	  //  // Brak przepływu na powrocie
	    
	  //   #nr := 7;
	  //   CASE "Tor1_alarmy".alarm[#nr].procedura OF
	            
	  //       2: //zalacz
	  //           IF "Tor1_obiekty".obiekt["C101FV11"].hmiPotwWysterowania =0 AND ("Tor1_hmi".button.bPauza.set=0)
	                
	                
	  //           THEN
	  //               IF "Tor1_alarmy".alarm[#nr].timerek < 32000 THEN
	  //                   "Tor1_alarmy".alarm[#nr].timerek := "Tor1_alarmy".alarm[#nr].timerek + 1;
	  //               END_IF;
	  //               "Tor1_alarmy".alarm[#nr].stan := BOOL_TO_INT("Tor1_alarmy".alarm[#nr].timerek >
	  //               "Tor1_RecepturyStacjaMycia".Receptura[#aktualnyNumerReceptury].Krok[#aktualnyKrokMycia].PM[4] * 10);
	  //           ELSE
	  //               "Tor1_alarmy".alarm[#nr].timerek := 0;
	  //               "Tor1_alarmy".alarm[#nr].stan := 0;
	  //           END_IF;
	            
	  //           IF "Tor1_alarmy".alarm[#nr].stan = 1
	  //               AND "Tor1_program".program.numerKroku <> 7700 THEN
	  //               "Tor1_hmi".button.bPauza.set := 1;
	  //               "krokZapauzowany" := "Tor1_program".program.numerKroku;
	  //               "Tor1_program".program.numerKroku := 7700;
	  //           END_IF;
	            
	  //       0:
	  //           "Tor1_alarmy".alarm[#nr].timerek := 0;
	  //           "Tor1_alarmy".alarm[#nr].stan := 0;
	            
	  //   END_CASE;
	    
	    
	    
	  //   //Niskie stężenie ługu
	    
	  //   #nr :=8;
	  //   CASE "Tor1_alarmy".alarm[#nr].procedura OF
	            
	  //       2: //zalacz
	  //           IF "Tor1_obiekty".obiekt["C101CT11"].WartośćPomiaru <=
	  //               0.5 * "Tor1_RecepturyStacjaMycia".Receptura[#aktualnyNumerReceptury].Krok[#aktualnyKrokMycia].PM[10]
	  //               AND #aktualnyKrokMycia=3
	                
	  //           THEN
	  //               IF "Tor1_alarmy".alarm[#nr].timerek < 32000 THEN
	  //                   "Tor1_alarmy".alarm[#nr].timerek := "Tor1_alarmy".alarm[#nr].timerek + 1;
	  //               END_IF;
	  //               "Tor1_alarmy".alarm[#nr].stan := BOOL_TO_INT("Tor1_alarmy".alarm[#nr].timerek >600);
	  //           ELSE
	  //               "Tor1_alarmy".alarm[#nr].timerek := 0;
	  //               "Tor1_alarmy".alarm[#nr].stan := 0;
	  //           END_IF;
	        
	            
	  //   END_CASE;
	    
	    
	    
	    
	  //   //Niskie stężenie kwasu
	    
	  //   #nr := 9;
	  //   CASE "Tor1_alarmy".alarm[#nr].procedura OF
	            
	  //       2: //zalacz
	  //           IF "Tor1_obiekty".obiekt["C101CT11"].WartośćPomiaru <=
	  //               0.5 * "Tor1_RecepturyStacjaMycia".Receptura[#aktualnyNumerReceptury].Krok[#aktualnyKrokMycia].PM[10]
	  //               AND #aktualnyKrokMycia=4
	                
	  //           THEN
	  //               IF "Tor1_alarmy".alarm[#nr].timerek < 32000 THEN
	  //                   "Tor1_alarmy".alarm[#nr].timerek := "Tor1_alarmy".alarm[#nr].timerek + 1;
	  //               END_IF;
	  //               "Tor1_alarmy".alarm[#nr].stan := BOOL_TO_INT("Tor1_alarmy".alarm[#nr].timerek > 600);
	  //           ELSE
	  //               "Tor1_alarmy".alarm[#nr].timerek := 0;
	  //               "Tor1_alarmy".alarm[#nr].stan := 0;
	  //           END_IF;
	            
	       
	            
	  //   END_CASE;
	    
	    
	  //   //Brak stężonego ługu
	    
	  //   #nr := 10;
	  //   CASE "Tor1_alarmy".alarm[#nr].procedura OF
	            
	  //       2: //zalacz
	  //           IF "CIP0_obiekty".obiekt["C2L1LL01"].hmiPotwWysterowania = 0
	                
	                
	                
	  //           THEN
	  //               IF "Tor1_alarmy".alarm[#nr].timerek < 32000 THEN
	  //                   "Tor1_alarmy".alarm[#nr].timerek := "Tor1_alarmy".alarm[#nr].timerek + 1;
	  //               END_IF;
	  //               "Tor1_alarmy".alarm[#nr].stan := BOOL_TO_INT("Tor1_alarmy".alarm[#nr].timerek > 600);
	  //           ELSE
	  //               "Tor1_alarmy".alarm[#nr].timerek := 0;
	  //               "Tor1_alarmy".alarm[#nr].stan := 0;
	  //           END_IF;
	            
	          
	            
	  //   END_CASE;
	    
	  //   //Brak stężonego kwasu
	    
	  //   #nr := 11;
	  //   CASE "Tor1_alarmy".alarm[#nr].procedura OF
	            
	  //       2: //zalacz
	  //           IF "CIP0_obiekty".obiekt["C2A1LL01"].hmiPotwWysterowania = 0
	                
	                
	                
	  //           THEN
	  //               IF "Tor1_alarmy".alarm[#nr].timerek < 32000 THEN
	  //                   "Tor1_alarmy".alarm[#nr].timerek := "Tor1_alarmy".alarm[#nr].timerek + 1;
	  //               END_IF;
	  //               "Tor1_alarmy".alarm[#nr].stan := BOOL_TO_INT("Tor1_alarmy".alarm[#nr].timerek > 600);
	  //           ELSE
	  //               "Tor1_alarmy".alarm[#nr].timerek := 0;
	  //               "Tor1_alarmy".alarm[#nr].stan := 0;
	  //           END_IF;
	    
	            
	  //   END_CASE;
	    
	    //Brak dezynfekanta
	    
	    #nr := 12;
	    CASE "Tor1_alarmy".alarm[#nr].procedura OF
	            
	        2: //zalacz
	            IF                "Cip".obiekt["Cip".tor[1].zbiorniczekDozowanieDezynfekantu.czujnikDolnegoPoziomu].hmiPotwWysterowania=0
	                OR (  "Cip".obiekt["Cip".tor[1].czujnikPrzepływuDozowanegoDezynfekantu].hmiPotwWysterowania=0
	                AND "Cip".obiekt["Cip".tor[1].zawórDozowaniaDezynfekantuwLinię].hmiPotwWysterowania=1)
	                
	            THEN
	                IF "Tor1_alarmy".alarm[#nr].timerek < 32000 THEN
	                    "Tor1_alarmy".alarm[#nr].timerek := "Tor1_alarmy".alarm[#nr].timerek + 1;
	                END_IF;
	                "Tor1_alarmy".alarm[#nr].stan := BOOL_TO_INT("Tor1_alarmy".alarm[#nr].timerek > 600);
	            ELSE
	                "Tor1_alarmy".alarm[#nr].timerek := 0;
	                "Tor1_alarmy".alarm[#nr].stan := 0;
	            END_IF;
	         
	    END_CASE;
	    
	    
	        
	  //       #nr := 13;
	  //       CASE "Tor1_alarmy".alarm[#nr].procedura OF
	                
	  //           2: //zalacz
	  //               IF  "Tor1_program".program.opóżnienie
	  //                   >"Tor1_RecepturyStacjaMycia".Receptura[#aktualnyNumerReceptury].Krok[#aktualnyKrokMycia].PM[19]
	                    
	                    
	  //               THEN
	  //                   IF "Tor1_alarmy".alarm[#nr].timerek < 32000 THEN
	  //                       "Tor1_alarmy".alarm[#nr].timerek := "Tor1_alarmy".alarm[#nr].timerek + 1;
	  //                   END_IF;
	  //                   "Tor1_alarmy".alarm[#nr].stan := BOOL_TO_INT("Tor1_alarmy".alarm[#nr].timerek > 600);
	  //               ELSE
	  //                   "Tor1_alarmy".alarm[#nr].timerek := 0;
	  //                   "Tor1_alarmy".alarm[#nr].stan := 0;
	  //               END_IF;
	         
	                
	  //       END_CASE;
	  
END_FUNCTION

FUNCTION "Tor1.procedury_obiektów" : Void
{ S7_Optimized_Access := 'TRUE' }
VERSION : 0.1
   VAR_TEMP 
      obj : Int;
      nr : Int;
      Mnr : String;
      aktualnyNumerReceptury : Int;
      aktualnyKrokMycia : Int;
      temp : Int;
   END_VAR


BEGIN
	    //program zawiera procedury dla napedów i zaworów dla procedur o numerze >1  (procedura 0 i 1 jest obsługiwana w programie Obsługa obiektów)
	    //procedury wyzwalane  z progrmu TablicaProcedór dla kolejnych kroków  "F1".obiekt["F100CP01"].procedura: = 2
	    //wyzwolenie procedury zero  automatycznie  wyłącza naped/zawór
	    //procedura:=1   uruchamia napęd/zawór na 100% - czyli załaczenie napedu jak kiedyś SET -- obsługiwana jest w programie Obsługa obiektów
	    //PAUZA może być obsługiwana w każdej procedurze z osobna
	    //
	    //open ctrl+shift+(*)Numeric
	    //close ctrl+shift+(/)Numeric
	    
	    #aktualnyNumerReceptury := "Tor1_RecepturyStacjaMycia".numerUżywanejReceptury;
	    #aktualnyKrokMycia := "Tor1_RecepturyStacjaMycia".numerKrokuMycia;
	    #temp := "Tor1_program".program.numerKroku;
	    
	    REGION POMPA PODAWANIA CIP
	    
	    #nr := "Cip".tor[1].pompaPodawaniaCip;
	    CASE "Tor1_program".program.numerKroku OF
	    7210, 7220, 7250:
	    "Cip".obiekt[#nr].procedura := 2;
	    7244, 7270, 7281..7287,7310, 7320,7321, 7414, 7420:
	    "Cip".obiekt[#nr].procedura := 3;
	    7240, 7242, 7243, 7246:
	    "Cip".obiekt[#nr].procedura := 6;
	    7100:
	    "Cip".obiekt[#nr].procedura := 7;
	    ELSE
	    "Cip".obiekt[#nr].procedura := 0;
	    
	    END_CASE;
	    
	    
	    
	    CASE "Cip".obiekt[#nr].procedura OF
	    2:
	    //wyzwolenie timerków
	    "Cip".obiekt[#nr].SetReset.czasDoSet := 3;
	    "Cip".obiekt[#nr].SetReset.inSet := "Cip".obiekt["Cip".tor[0].zbiornikwodyCzystej.czujnikDolnegoPoziomu].hmiPotwWysterowania
	    OR "Cip".obiekt["Cip".tor[0].zbiornikWodyWtórnej.czujnikDolnegoPoziomu].hmiPotwWysterowania;
	    "Cip".obiekt[#nr].SetReset.czasDoReset := 5;
	    "Cip".obiekt[#nr].SetReset.inReset := (NOT "Cip".obiekt["Cip".tor[0].zbiornikwodyCzystej.czujnikDolnegoPoziomu].hmiPotwWysterowania
	    AND NOT "Cip".obiekt["Cip".tor[0].zbiornikWodyWtórnej.czujnikDolnegoPoziomu].hmiPotwWysterowania) OR
	    ("Cip".obiekt["Cip".tor[1].zbiornikDezynfekantu.czujnikDolnegoPoziomu].hmiPotwWysterowania = 0 AND ("Tor1_program".program.numerKroku = 7282
	    OR "Tor1_program".program.numerKroku = 7283))
	    
	    ;
	    
	    //załaczanie
	    "Cip".obiekt[#nr].inStartAuto := "Cip".obiekt[#nr].SetReset.wyjście;
	    
	    //wysterowanie
	    "Cip".obiekt[#nr].inZadaneWysterowanieAuto :=  //pid_out wypełniamy w wywołaniu pida z out pida
	    LIMIT(IN := "Cip".obiekt[#nr].pid_Out, MN := 0.0, MX := 100.0);//pid_out ;
	    
	    ////PID
	    "Cip".obiekt[#nr].pid_SP := "Tor1_RecepturyStacjaMycia".Receptura[#aktualnyNumerReceptury].Krok[#aktualnyKrokMycia].PM[2];
	    "Cip".obiekt[#nr].pid_PV := "Cip".obiekt["Cip".tor[1].przepływomierzZaWymiennikiem].WartośćPomiaru;
	    
	    
	    3: //wyzwolenie timerków
	    
	    //wyzwolenie timerków
	    "Cip".obiekt[#nr].SetReset.czasDoSet := 3;
	    "Cip".obiekt[#nr].SetReset.inSet := "Cip".obiekt["Cip".tor[0].zbiornikwodyCzystej.czujnikDolnegoPoziomu].hmiPotwWysterowania
	    ;
	    "Cip".obiekt[#nr].SetReset.czasDoReset := 5;
	    "Cip".obiekt[#nr].SetReset.inReset := NOT "Cip".obiekt["Cip".tor[0].zbiornikwodyCzystej.czujnikDolnegoPoziomu].hmiPotwWysterowania
	    ;
	    //załaczanie
	    
	    "Cip".obiekt[#nr].inStartAuto := "Cip".obiekt[#nr].SetReset.wyjście;
	    
	    //wysterowanie
	    "Cip".obiekt[#nr].inZadaneWysterowanieAuto :=  //pid_out wypełniamy w wywołaniu pida z out pida
	    LIMIT(IN := "Cip".obiekt[#nr].pid_Out, MN := 0.0, MX := 100.0);//pid_out ;
	    
	    ////PID
	    "Cip".obiekt[#nr].pid_SP := "Tor1_RecepturyStacjaMycia".Receptura[#aktualnyNumerReceptury].Krok[#aktualnyKrokMycia].PM[2];
	    "Cip".obiekt[#nr].pid_PV := "Cip".obiekt["Cip".tor[1].przepływomierzZaWymiennikiem].WartośćPomiaru;
	    
	    4: //wyzwolenie timerków
	    
	    //wyzwolenie timerków
	    "Cip".obiekt[#nr].SetReset.czasDoSet := 3;
	    "Cip".obiekt[#nr].SetReset.inSet :=
	    "Cip".obiekt["Cip".tor[0].zbiornikwodyCzystej.czujnikDolnegoPoziomu].hmiPotwWysterowania
	    AND #aktualnyKrokMycia = 3
	    ;
	    "Cip".obiekt[#nr].SetReset.czasDoReset := 5;
	    "Cip".obiekt[#nr].SetReset.inReset :=
	    NOT "Cip".obiekt["Cip".tor[0].zbiornikwodyCzystej.czujnikDolnegoPoziomu].hmiPotwWysterowania
	    AND #aktualnyKrokMycia = 3
	    ;
	    //załaczanie
	    "Cip".obiekt[#nr].inStartAuto := "Cip".obiekt[#nr].SetReset.wyjście;
	    
	    //wysterowanie
	    "Cip".obiekt[#nr].inZadaneWysterowanieAuto :=  //pid_out wypełniamy w wywołaniu pida z out pida
	    LIMIT(IN := "Cip".obiekt[#nr].pid_Out, MN := 0.0, MX := 100.0);//pid_out ;
	    
	    ////PID
	    "Cip".obiekt[#nr].pid_SP := "Tor1_RecepturyStacjaMycia".Receptura[#aktualnyNumerReceptury].Krok[#aktualnyKrokMycia].PM[2];
	    "Cip".obiekt[#nr].pid_PV := "Cip".obiekt["Cip".tor[1].przepływomierzZaWymiennikiem].WartośćPomiaru;
	    
	    5: //wyzwolenie timerków
	    
	    //wyzwolenie timerków
	    "Cip".obiekt[#nr].SetReset.czasDoSet := 3;
	    "Cip".obiekt[#nr].SetReset.inSet := "Cip".obiekt["Cip".tor[0].zbiornikwodyCzystej.czujnikDolnegoPoziomu].hmiPotwWysterowania
	    AND #aktualnyKrokMycia = 4
	    ;
	    "Cip".obiekt[#nr].SetReset.czasDoReset := 5;
	    "Cip".obiekt[#nr].SetReset.inReset := NOT "Cip".obiekt["Cip".tor[0].zbiornikwodyCzystej.czujnikDolnegoPoziomu].hmiPotwWysterowania
	    AND #aktualnyKrokMycia = 4
	    ;
	    //załaczanie
	    "Cip".obiekt[#nr].inStartAuto := "Cip".obiekt[#nr].SetReset.wyjście;
	    
	    //wysterowanie
	    "Cip".obiekt[#nr].inZadaneWysterowanieAuto :=  //pid_out wypełniamy w wywołaniu pida z out pida
	    LIMIT(IN := "Cip".obiekt[#nr].pid_Out, MN := 0.0, MX := 100.0);//pid_out ;
	    
	    ////PID
	    "Cip".obiekt[#nr].pid_SP := "Tor1_RecepturyStacjaMycia".Receptura[#aktualnyNumerReceptury].Krok[#aktualnyKrokMycia].PM[2];
	    "Cip".obiekt[#nr].pid_PV := "Cip".obiekt["Cip".tor[1].przepływomierzZaWymiennikiem].WartośćPomiaru;
	    
	    6: //wyzwolenie timerków
	    //wyzwolenie timerków
	    "Cip".obiekt[#nr].SetReset.czasDoSet := 3;
	    "Cip".obiekt[#nr].SetReset.inSet :=
	    ("Cip".obiekt["Cip".tor[0].zbiornikwodyCzystej.czujnikDolnegoPoziomu].hmiPotwWysterowania
	    AND #aktualnyKrokMycia = 4)
	    OR
	    ("Cip".obiekt["Cip".tor[0].zbiornikwodyCzystej.czujnikDolnegoPoziomu].hmiPotwWysterowania
	    AND #aktualnyKrokMycia = 3)
	    ;
	    "Cip".obiekt[#nr].SetReset.czasDoReset := 5;
	    "Cip".obiekt[#nr].SetReset.inReset :=
	    (NOT "Cip".obiekt["Cip".tor[0].zbiornikwodyCzystej.czujnikDolnegoPoziomu].hmiPotwWysterowania
	    AND #aktualnyKrokMycia = 4)
	    OR
	    (NOT "Cip".obiekt["Cip".tor[0].zbiornikwodyCzystej.czujnikDolnegoPoziomu].hmiPotwWysterowania
	    AND #aktualnyKrokMycia = 3);
	    
	    //załaczanie
	    "Cip".obiekt[#nr].inStartAuto := 1;
	    
	    //wysterowanie
	    "Cip".obiekt[#nr].inZadaneWysterowanieAuto :=  //pid_out wypełniamy w wywołaniu pida z out pida
	    LIMIT(IN := "Cip".obiekt[#nr].pid_Out, MN := 0.0, MX := 100.0);//pid_out ;
	    
	    ////PID
	    "Cip".obiekt[#nr].pid_SP := "Tor1_RecepturyStacjaMycia".Receptura[#aktualnyNumerReceptury].Krok[#aktualnyKrokMycia].PM[2];
	    "Cip".obiekt[#nr].pid_PV := "Cip".obiekt["Cip".tor[1].przepływomierzZaWymiennikiem].WartośćPomiaru;
	    
	    
	    7:
	    //wyzwolenie timerków
	    "Cip".obiekt[#nr].SetReset.czasDoSet := 1;
	    "Cip".obiekt[#nr].SetReset.inSet :=
	    "Cip".obiekt["Cip".tor[2].pompaPodawaniaCip].inStartAuto; //cpNiex
	    
	    "Cip".obiekt[#nr].SetReset.czasDoReset := 1;
	    "Cip".obiekt[#nr].SetReset.inReset :=
	    NOT "Cip".obiekt["Cip".tor[2].pompaPodawaniaCip].inStartAuto; //cpNiex
	    //załaczanie
	    "Cip".obiekt[#nr].inStartAuto := "Cip".obiekt[#nr].SetReset.wyjście;
	    //wysterowanie
	    "Cip".obiekt[#nr].inZadaneWysterowanieAuto := 100.0;
	    
	    
	    
	    0:
	    ;
	    
	    // resetowanie całkującej części regulatora aby nie przejebać temperatury
	    // "PID_Compact23".IntegralResetMode := 3;
	    // "PID_Compact23".OverwriteInitialOutputValue := "F1.SP"."203"- 1.0;
	    // "PID_Compact23".Reset := "F1".obiekt["F100LT01"].WartośćPomiaru > 70.0;
	    // := LIMIT(IN := "APA".obiekt["PID123"].outWysterowanieUrządzenia,
	    // MN := 0.0, MX := "APA".obiekt["H101TT01"].WartośćPomiaru + "H1.STP"."214");
	    
	    END_CASE;
	    
	    IF "Cip".obiekt[#nr].procedura > 0 THEN
	    
	        IF "Cip".obiekt[#nr].inStartAuto = 0 THEN
	            "Cip".obiekt[#nr].inZadaneWysterowanieAuto := 0.0;
	            "Cip".obiekt[#nr].pid_SP := 0.0;
	        END_IF;
	    END_IF;
	    
	    
	    "PID.pompaPodawaniaCipTor1"(Setpoint := "Cip".obiekt[#nr].pid_SP,
	                        Input := "Cip".obiekt[#nr].pid_PV,
	                        Reset := "Cip".obiekt[#nr].hmiResetAwaria,
	                        Output => "Cip".obiekt[#nr].pid_Out);
	    "PID.pompaPodawaniaCipTor1".Retain.CtrlParams.Gain := 1.2;
	    "PID.pompaPodawaniaCipTor1".Retain.CtrlParams.Ti := 3;
	    "PID.pompaPodawaniaCipTor1".Retain.CtrlParams.Td := 0.1;
	    
	    
	    
	    "PID.pompaPodawaniaCipTor1".IntegralResetMode := 3;
	    "PID.pompaPodawaniaCipTor1".OverwriteInitialOutputValue := 1;
	    "PID.pompaPodawaniaCipTor1".Reset := (
	    "Cip".obiekt[#nr].procedura = 0 OR "Cip".obiekt[#nr].inStartAuto = 0
	    OR "numer_kroku_stary_1" <> "Tor1_program".program.numerKroku);
	    
	    "numer_kroku_stary_1" := "Tor1_program".program.numerKroku;
	    END_REGION
	    
	    REGION POMPA PRZYGOTOWANIA CIP(DRUGA PODAWCZA)
	    
	    //pompa powrotu/ Program musi ustalić, który tor myje stacje,
	    //drugi staje się pompą powrotu (staje się pompą 102 - tymczasowo)
	    //obsługa wykrywania w CIP1_wejściach_wyjściach
	    #nr := "Cip".tor[2].pompaPodawaniaCip;
	    CASE "Tor1_program".program.numerKroku OF
	    7401..7404, 7410..7414:
	    "Cip".obiekt[#nr].procedura := 2
	    ;
	    7230..7440:
	    "Cip".obiekt[#nr].procedura := 3;
	    7450, 7460:
	    "Cip".obiekt[#nr].procedura := 4;
	    ELSE
	    "Cip".obiekt[#nr].procedura := 0;
	    
	    END_CASE;
	    
	    
	    CASE "Cip".obiekt[#nr].procedura OF
	    2:
	    //wyzwolenie timerków
	    "Cip".obiekt[#nr].SetReset.czasDoSet := 3;
	    "Cip".obiekt[#nr].SetReset.inSet :=
	    "Cip".obiekt["Cip".tor[0].zbiornikWodyWtórnej.czujnikDolnegoPoziomu].hmiPotwWysterowania;
	    
	    "Cip".obiekt[#nr].SetReset.czasDoReset := 60;
	    "Cip".obiekt[#nr].SetReset.inReset :=
	    NOT "Cip".obiekt["Cip".tor[0].zbiornikWodyWtórnej.czujnikDolnegoPoziomu].hmiPotwWysterowania;
	    //załaczanie
	    
	    "Cip".obiekt[#nr].inStartAuto := "Cip".obiekt[#nr].SetReset.wyjście;
	    
	    //wysterowanie
	    "Cip".obiekt[#nr].inZadaneWysterowanieAuto := 100.0;
	    
	    3:
	    //wyzwolenie timerków
	    "Cip".obiekt[#nr].SetReset.czasDoSet := 3;
	    "Cip".obiekt[#nr].SetReset.inSet :=
	    "Cip".obiekt["Cip".tor[0].zbiornikŁugu.czujnikDolnegoPoziomu].hmiPotwWysterowania;
	    
	    "Cip".obiekt[#nr].SetReset.czasDoReset := 60;
	    "Cip".obiekt[#nr].SetReset.inReset :=
	    NOT "Cip".obiekt["Cip".tor[0].zbiornikŁugu.czujnikDolnegoPoziomu].hmiPotwWysterowania;
	    //załaczanie
	    
	    "Cip".obiekt[#nr].inStartAuto := "Cip".obiekt[#nr].SetReset.wyjście;
	    
	    //wysterowanie
	    "Cip".obiekt[#nr].inZadaneWysterowanieAuto := 100.0;
	    4:
	    //wyzwolenie timerków
	    "Cip".obiekt[#nr].SetReset.czasDoSet := 3;
	    "Cip".obiekt[#nr].SetReset.inSet :=
	    "Cip".obiekt["Cip".tor[0].zbiornikKwasu.czujnikDolnegoPoziomu].hmiPotwWysterowania;
	    
	    "Cip".obiekt[#nr].SetReset.czasDoReset := 60;
	    "Cip".obiekt[#nr].SetReset.inReset :=
	    NOT "Cip".obiekt["Cip".tor[0].zbiornikKwasu.czujnikDolnegoPoziomu].hmiPotwWysterowania;
	    //załaczanie
	    "Cip".obiekt[#nr].inStartAuto := "Cip".obiekt[#nr].SetReset.wyjście;
	    //wysterowanie
	    "Cip".obiekt[#nr].inZadaneWysterowanieAuto := 100.0;
	    
	    
	    
	    END_CASE;
	    
	    END_REGION
	    
	    REGION ZAWÓR DOZOWANIA ŁUGU W LINIE
	    
	        #nr := "Cip".tor[0].zawórDozowaniaLuguwLinię;
	        
	        CASE "Tor1_program".program.numerKroku OF
	            7243, 7320:
	                "Cip".obiekt[#nr].procedura := 3;
	            ELSE
	                "Cip".obiekt[#nr].procedura := 0;
	                "Cip".obiekt[#nr].Flipaj.in := 0;
	        END_CASE;
	        
	    CASE "Cip".obiekt[#nr].procedura OF
	    2:
	    //set - warunki dla wejścia funkcji Set
	    "Cip".obiekt[#nr].SetReset.czasDoSet := 10;
	    "Cip".obiekt[#nr].SetReset.inSet :=
	    "Cip".obiekt["Cip".tor[0].zbiorniczekDozowaniaŁugu.czujnikDolnegoPoziomu].hmiPotwWysterowania = 1
	    AND #aktualnyKrokMycia = 3;
	    
	    //reset - warunki dla wejścia funkcji Reset
	    "Cip".obiekt[#nr].SetReset.czasDoReset := 0;
	    "Cip".obiekt[#nr].SetReset.inReset :=
	    "Cip".obiekt["Cip".tor[0].zbiorniczekDozowaniaŁugu.czujnikDolnegoPoziomu].hmiPotwWysterowania = 0
	    OR #aktualnyKrokMycia = 4;
	    
	    //załaczanie
	    "Cip".obiekt[#nr].Flipaj.czas_ON := 300;
	    "Cip".obiekt[#nr].Flipaj.czas_OFF := 100;
	    "Cip".obiekt[#nr].Flipaj.ile_petli := 999;
	    "Cip".obiekt[#nr].Flipaj.in := "Cip".obiekt[#nr].SetReset.wyjście;
	    "Cip".obiekt[#nr].inStartAuto := "Cip".obiekt[#nr].Flipaj.Q;
	    
	    //wysterowanie
	    "Cip".obiekt[#nr].inZadaneWysterowanieAuto := 100.0;
	    
	    3:
	    //set - warunki dla wejścia funkcji Set
	    "Cip".obiekt[#nr].SetReset.czasDoSet := 10;
	    "Cip".obiekt[#nr].SetReset.inSet :=
	    "Cip".obiekt["Cip".tor[0].zbiorniczekDozowaniaŁugu.czujnikDolnegoPoziomu].hmiPotwWysterowania = 1
	    AND ("Tor1_RecepturyStacjaMycia".numerKrokuMycia = 3)
	    AND ("Cip".obiekt["Cip".tor[1].przewodnośćNaPowrocie].WartośćPomiaru <
	    "Tor1_RecepturyStacjaMycia".Receptura[#aktualnyNumerReceptury].Krok[#aktualnyKrokMycia].PM[11]);
	    
	    //reset - warunki dla wejścia funkcji Reset
	    "Cip".obiekt[#nr].SetReset.czasDoReset := 0;
	    "Cip".obiekt[#nr].SetReset.inReset :=
	    "Cip".obiekt["Cip".tor[0].zbiorniczekDozowaniaŁugu.czujnikDolnegoPoziomu].hmiPotwWysterowania = 0
	    OR ("Tor1_RecepturyStacjaMycia".numerKrokuMycia = 4)
	    OR ("Cip".obiekt["Cip".tor[1].przewodnośćNaPowrocie].WartośćPomiaru >=
	    "Tor1_RecepturyStacjaMycia".Receptura[#aktualnyNumerReceptury].Krok[#aktualnyKrokMycia].PM[11]);
	    
	    //załaczanie
	    "Cip".obiekt[#nr].Flipaj.czas_ON := REAL_TO_INT(
	                                                    "Tor1_RecepturyStacjaMycia".
	                                                    Receptura[#aktualnyNumerReceptury].
	                                                    Krok[#aktualnyKrokMycia].PM[26] * 10);
	    "Cip".obiekt[#nr].Flipaj.czas_OFF := REAL_TO_INT(
	                                                     "Tor1_RecepturyStacjaMycia".
	                                                     Receptura[#aktualnyNumerReceptury].
	                                                     Krok[#aktualnyKrokMycia].PM[27] * 10);
	    "Cip".obiekt[#nr].Flipaj.ile_petli :=
	    REAL_TO_INT("Tor1_RecepturyStacjaMycia".Receptura[#aktualnyNumerReceptury].Krok[#aktualnyKrokMycia].PM[20] /
	                ("Tor1_RecepturyStacjaMycia".Receptura[#aktualnyNumerReceptury].Krok[#aktualnyKrokMycia].PM[26] +
	                "Tor1_RecepturyStacjaMycia".Receptura[#aktualnyNumerReceptury].Krok[#aktualnyKrokMycia].PM[27] + 1.0));
	    "Cip".obiekt[#nr].Flipaj.in := "Cip".obiekt[#nr].SetReset.wyjście;
	    "Cip".obiekt[#nr].inStartAuto := "Cip".obiekt[#nr].Flipaj.Q;
	    
	    //wysterowanie
	    "Cip".obiekt[#nr].inZadaneWysterowanieAuto := 100.0;
	0:
	    "Cip".obiekt[#nr].Flipaj.in := 0;
	    END_CASE;
	    END_REGION
	    
	    REGION ZAWÓR DOZOWANIA KWASU W LINIE
	    
	        #nr := "Cip".tor[0].zawórDozowaniaKwasuwLinię;
	        
	        CASE "Tor1_program".program.numerKroku OF
	            7243, 7320:
	                "Cip".obiekt[#nr].procedura := 3;
	            ELSE
	                "Cip".obiekt[#nr].procedura := 0;
	                "Cip".obiekt[#nr].Flipaj.in := 0;
	        END_CASE;
	        
	    CASE "Cip".obiekt[#nr].procedura OF
	    2:
	    //set - warunki dla wejścia funkcji Set
	    "Cip".obiekt[#nr].SetReset.czasDoSet := 10;
	    "Cip".obiekt[#nr].SetReset.inSet :=
	    "Cip".obiekt["Cip".tor[0].zbiorniczekDozowaniaKwasu.czujnikDolnegoPoziomu].hmiPotwWysterowania = 1
	    AND ("Tor1_RecepturyStacjaMycia".numerKrokuMycia = 4);
	    
	    //reset - warunki dla wejścia funkcji Reset
	    "Cip".obiekt[#nr].SetReset.czasDoReset := 0;
	    "Cip".obiekt[#nr].SetReset.inReset :=
	    "Cip".obiekt["Cip".tor[0].zbiorniczekDozowaniaKwasu.czujnikDolnegoPoziomu].hmiPotwWysterowania = 0
	    OR ("Tor1_RecepturyStacjaMycia".numerKrokuMycia = 3);
	    
	    //załaczanie
	    "Cip".obiekt[#nr].Flipaj.czas_ON := 300;
	    "Cip".obiekt[#nr].Flipaj.czas_OFF := 100;
	    "Cip".obiekt[#nr].Flipaj.ile_petli := 999;
	    "Cip".obiekt[#nr].Flipaj.in := "Cip".obiekt[#nr].SetReset.wyjście;
	    "Cip".obiekt[#nr].inStartAuto := "Cip".obiekt[#nr].Flipaj.Q;
	    
	    //wysterowanie
	    "Cip".obiekt[#nr].inZadaneWysterowanieAuto := 100.0;
	    
	    3:
	    //set - warunki dla wejścia funkcji Set
	    "Cip".obiekt[#nr].SetReset.czasDoSet := 100;
	    "Cip".obiekt[#nr].SetReset.inSet :=
	    "Cip".obiekt["Cip".tor[0].zbiorniczekDozowaniaKwasu.czujnikDolnegoPoziomu].hmiPotwWysterowania = 1
	    AND ("Tor1_RecepturyStacjaMycia".numerKrokuMycia = 4) //warunki dla toru Cip1
	    AND ("Cip".obiekt["Cip".tor[1].przewodnośćNaPowrocie].WartośćPomiaru <
	    "Tor1_RecepturyStacjaMycia".Receptura[#aktualnyNumerReceptury].Krok[#aktualnyKrokMycia].PM[11]);
	    
	    
	    //reset - warunki dla wejścia funkcji Reset
	    "Cip".obiekt[#nr].SetReset.czasDoReset := 0;
	    "Cip".obiekt[#nr].SetReset.inReset :=
	    "Cip".obiekt["Cip".tor[0].zbiorniczekDozowaniaKwasu.czujnikDolnegoPoziomu].hmiPotwWysterowania = 0
	    OR ("Tor1_RecepturyStacjaMycia".numerKrokuMycia = 3) //warunki dla toru Cip1
	    OR ("Cip".obiekt["Cip".tor[1].przewodnośćNaPowrocie].WartośćPomiaru >=
	    "Tor1_RecepturyStacjaMycia".Receptura[#aktualnyNumerReceptury].Krok[#aktualnyKrokMycia].PM[11]);
	    
	    //załaczanie
	    "Cip".obiekt[#nr].Flipaj.czas_ON := REAL_TO_INT(
	                                                    "Tor1_RecepturyStacjaMycia".
	                                                    Receptura[#aktualnyNumerReceptury].
	                                                    Krok[#aktualnyKrokMycia].PM[26] * 10);
	    "Cip".obiekt[#nr].Flipaj.czas_OFF := REAL_TO_INT(
	                                                     "Tor1_RecepturyStacjaMycia".
	                                                     Receptura[#aktualnyNumerReceptury].
	                                                     Krok[#aktualnyKrokMycia].PM[27] * 10);
	    "Cip".obiekt[#nr].Flipaj.ile_petli :=
	    REAL_TO_INT("Tor1_RecepturyStacjaMycia".Receptura[#aktualnyNumerReceptury].Krok[#aktualnyKrokMycia].PM[20] /
	                ("Tor1_RecepturyStacjaMycia".Receptura[#aktualnyNumerReceptury].Krok[#aktualnyKrokMycia].PM[26] +
	                "Tor1_RecepturyStacjaMycia".Receptura[#aktualnyNumerReceptury].Krok[#aktualnyKrokMycia].PM[27] + 1.0));
	    "Cip".obiekt[#nr].Flipaj.in := "Cip".obiekt[#nr].SetReset.wyjście;
	    "Cip".obiekt[#nr].inStartAuto := "Cip".obiekt[#nr].Flipaj.Q;
	    
	    //wysterowanie
	    "Cip".obiekt[#nr].inZadaneWysterowanieAuto := 100.0;
	0:
	    "Cip".obiekt[#nr].Flipaj.in := 0;
	    END_CASE;
	    
	    END_REGION
	    
	    REGION POMPKA DOZOWANIA DEZYNFEKANTU W LINIE
	    
	        #nr := "Cip".tor[1].pompkaDozowaniaDezynfekantuwLinię;
	        
	        CASE "Tor1_program".program.numerKroku OF
	            7282:
	                "Cip".obiekt[#nr].procedura := 2;
	            ELSE
	                "Cip".obiekt[#nr].procedura := 0;
	        END_CASE;
	        
	    CASE "Cip".obiekt[#nr].procedura OF
	    2:
	    
	    //
	    //załaczanie
	    "Cip".obiekt[#nr].Flipaj.czas_ON := REAL_TO_INT(
	                                                  "Tor1_RecepturyStacjaMycia".
	                                                  Receptura[#aktualnyNumerReceptury].
	                                                  Krok[#aktualnyKrokMycia].PM[26] * 10);
	    "Cip".obiekt[#nr].Flipaj.czas_OFF := REAL_TO_INT(
	                                                   "Tor1_RecepturyStacjaMycia".
	                                                   Receptura[#aktualnyNumerReceptury].
	                                                   Krok[#aktualnyKrokMycia].PM[27] * 10);
	  "Cip".obiekt[#nr].Flipaj.ile_petli := 999;
	    // REAL_TO_INT("Tor1_RecepturyStacjaMycia".Receptura[#aktualnyNumerReceptury].Krok[#aktualnyKrokMycia].PM[20] /
	    //             ("Tor1_RecepturyStacjaMycia".Receptura[#aktualnyNumerReceptury].Krok[#aktualnyKrokMycia].PM[26] +
	    //             "Tor1_RecepturyStacjaMycia".Receptura[#aktualnyNumerReceptury].Krok[#aktualnyKrokMycia].PM[27] + 1.0));
	    
	    ;
	    "Cip".obiekt[#nr].Flipaj.in := 1;
	    "Cip".obiekt[#nr].inStartAuto := "Cip".obiekt[#nr].Flipaj.Q;
	    
	    "Cip".obiekt[#nr].inStartAuto := "Cip".obiekt[#nr].Flipaj.Q;
	    0:
	    "Cip".obiekt[#nr].Flipaj.in := 0;
	    END_CASE;
	END_REGION
	REGION zawor  DOZOWANIA DEZYNFEKANTU W LINIE
	    
	    #nr := "Cip".tor[1].zawórDozowaniaDezynfekantuwLinię;
	    
	    CASE "Tor1_program".program.numerKroku OF
	        7282:
	            "Cip".obiekt[#nr].procedura := 2;
	        ELSE
	            "Cip".obiekt[#nr].procedura := 0;
	    END_CASE;
	    
	    CASE "Cip".obiekt[#nr].procedura OF
	        2:
	            
	            //
	            //załaczanie
	      
	            
	            ;
	           
	            "Cip".obiekt[#nr].inStartAuto := "Cip".obiekt["Cip".tor[1].pompkaDozowaniaDezynfekantuwLinię].outStartUrządzenie;
	      
	        0:
	            "Cip".obiekt[#nr].Flipaj.in := 0;
	    END_CASE;
	END_REGION
	    
	    REGION ZAWOR ZRZUTOWY DO KANALIZACJI
	    
	    
	    #nr := "Cip".tor[1].zawórZrzutowyDoKanalizacji;
	    CASE "Tor1_program".program.numerKroku OF
	    7100, 7202..7246, 7270,7287,7310, 7320, 7321, 7402, 7403, 7411..7414, 7420, 7431..7435, 7440, 7460:
	    "Cip".obiekt[#nr].procedura := 2;
	  
	    ELSE
	    "Cip".obiekt[#nr].procedura := 0;
	    
	    END_CASE;
	    
	    CASE "Cip".obiekt[#nr].procedura OF
	    2:
	    //wyzwolenie timerków
	    "Cip".obiekt[#nr].SetReset.czasDoSet := 2;
	    "Cip".obiekt[#nr].SetReset.inSet :=
	    "Cip".obiekt["Cip".tor[1].zawórPowrotnyWodyWtórnej].outStartUrządzenie
	    OR "Cip".obiekt["Cip".tor[1].zawórPowrotnyŁugu].outStartUrządzenie
	    OR "Cip".obiekt["Cip".tor[1].zawórPowrotnyKwasu].outStartUrządzenie;
	    
	    "Cip".obiekt[#nr].SetReset.czasDoReset := 2;
	    "Cip".obiekt[#nr].SetReset.inReset :=
	    NOT "Cip".obiekt["Cip".tor[1].zawórPowrotnyWodyWtórnej].outStartUrządzenie
	    AND NOT "Cip".obiekt["Cip".tor[1].zawórPowrotnyŁugu].outStartUrządzenie
	    AND NOT "Cip".obiekt["Cip".tor[1].zawórPowrotnyKwasu].outStartUrządzenie;
	    //załaczanie
	    "Cip".obiekt[#nr].inStartAuto := "Cip".obiekt[#nr].SetReset.wyjście;
	    
	    3:
	    //wyzwolenie timerków
	    "Cip".obiekt[#nr].SetReset.czasDoSet := 2;
	    "Cip".obiekt[#nr].SetReset.inSet :=
	    "Cip".obiekt["Cip".tor[1].zawórBypassPrzygotowaniaStacji].outStartUrządzenie;
	    
	    
	    "Cip".obiekt[#nr].SetReset.czasDoReset := 2;
	    "Cip".obiekt[#nr].SetReset.inReset :=
	    NOT "Cip".obiekt["Cip".tor[1].zawórBypassPrzygotowaniaStacji].outStartUrządzenie;
	    
	    //załaczanie
	    "Cip".obiekt[#nr].inStartAuto := "Cip".obiekt[#nr].SetReset.wyjście;
	    END_CASE;
	    END_REGION
	    
	    REGION ZAWOR WYDAWCZY CIP
	    
	    #nr := "Cip".tor[1].zawórWydawczyCip;
	    CASE "Tor1_program".program.numerKroku OF
	    7210..7290:
	    "Cip".obiekt[#nr].procedura := 1;
	    
	    ELSE
	    "Cip".obiekt[#nr].procedura := 0;
	    
	    END_CASE;
	    
	    CASE "Cip".obiekt[#nr].procedura OF
	    2:
	    //wyzwolenie timerków
	    "Cip".obiekt[#nr].SetReset.czasDoSet := 2;
	    "Cip".obiekt[#nr].SetReset.inSet :=
	    "Cip".obiekt["Cip".tor[1].pompaPodawaniaCip].outStartUrządzenie;
	    
	    "Cip".obiekt[#nr].SetReset.czasDoReset := 2;
	    "Cip".obiekt[#nr].SetReset.inReset :=
	    NOT "Cip".obiekt["Cip".tor[1].pompaPodawaniaCip].outStartUrządzenie;
	    //załaczanie
	    "Cip".obiekt[#nr].inStartAuto := "Cip".obiekt[#nr].SetReset.wyjście;
	    
	    END_CASE;
	    END_REGION
	    
	    REGION ZAWOR BYPASS PRZYGOTOWANIA STACJI
	    
	    #nr := "Cip".tor[1].zawórBypassPrzygotowaniaStacji;
	    CASE "Tor1_program".program.numerKroku OF
	    7210..7290:
	    "Cip".obiekt[#nr].procedura := 2;
	    7320:
	    "Cip".obiekt[#nr].procedura := 3;
	    ELSE
	    "Cip".obiekt[#nr].procedura := 0;
	    
	    END_CASE;
	    CASE "Cip".obiekt[#nr].procedura OF
	    2:
	    //wyzwolenie timerków
	    "Cip".obiekt[#nr].SetReset.czasDoSet := 2;
	    "Cip".obiekt[#nr].SetReset.inSet :=NOT 
	    "Cip".obiekt["Cip".tor[1].zawórWydawczyCip].outStartUrządzenie;
	    
	    "Cip".obiekt[#nr].SetReset.czasDoReset := 2;
	    "Cip".obiekt[#nr].SetReset.inReset :=
	  "Cip".obiekt["Cip".tor[1].zawórWydawczyCip].outStartUrządzenie;
	    //załaczanie
	    "Cip".obiekt[#nr].inStartAuto := "Cip".obiekt[#nr].SetReset.wyjście;
	    3:
	    
	    //załaczanie
	    "Cip".obiekt[#nr].inStartAuto := 1;
	    
	    END_CASE;
	    END_REGION
	    
	    REGION ZAWOR WYDAWCZY WODY WTORNEJ
	    
	    #nr := "Cip".tor[1].zawórWydawczyWodyWtórnej;
	    
	    CASE "Tor1_program".program.numerKroku OF
	    7210,7230:
	    "Cip".obiekt[#nr].procedura := 2;
	    7100:
	    "Cip".obiekt[#nr].procedura := 3;
	    ELSE
	    "Cip".obiekt[#nr].procedura := 0;
	    
	    END_CASE;
	    
	    
	    
	    CASE "Cip".obiekt[#nr].procedura OF
	    2:
	    //wyzwolenie timerków
	    "Cip".obiekt[#nr].SetReset.czasDoSet := 3;
	    "Cip".obiekt[#nr].SetReset.inSet :=
	    "Cip".obiekt["Cip".tor[0].zbiornikWodyWtórnej.czujnikDolnegoPoziomu].hmiPotwWysterowania
	    AND (#aktualnyKrokMycia = 1 OR #aktualnyKrokMycia = 2);
	    
	    "Cip".obiekt[#nr].SetReset.czasDoReset := 10;
	    "Cip".obiekt[#nr].SetReset.inReset :=
	    NOT "Cip".obiekt["Cip".tor[0].zbiornikWodyWtórnej.czujnikDolnegoPoziomu].hmiPotwWysterowania
	    OR (#aktualnyKrokMycia <> 1 AND #aktualnyKrokMycia <> 2);
	    //załaczanie
	    "Cip".obiekt[#nr].inStartAuto := "Cip".obiekt[#nr].SetReset.wyjście;
	    3:
	    //wyzwolenie timerków
	    "Cip".obiekt[#nr].SetReset.czasDoSet := 3;
	    "Cip".obiekt[#nr].SetReset.inSet :=
	    ("Tor2_program".program.numerKroku >= 7401 AND
	    "Tor2_program".program.numerKroku <= 7420);
	    
	    
	    "Cip".obiekt[#nr].SetReset.czasDoReset := 60;
	    "Cip".obiekt[#nr].SetReset.inReset :=
	    NOT ("Tor2_program".program.numerKroku >= 7401 AND
	    "Tor2_program".program.numerKroku <= 7420);
	    
	    //załaczanie
	    "Cip".obiekt[#nr].inStartAuto := "Cip".obiekt[#nr].SetReset.wyjście;
	    
	    END_CASE;
	    END_REGION
	    
	    REGION ZAWÓR POWROTNY WODY WTORNEJ
	    
	    #nr := "Cip".tor[1].zawórPowrotnyWodyWtórnej;
	    CASE "Tor1_program".program.numerKroku OF
	        7250, 7270, 7285, 7287:
	            "Cip".obiekt[#nr].procedura := 2;
	        7402, 7403, 7411, 7414, 7420:
	            "Cip".obiekt[#nr].procedura := 1;
	        ELSE
	            "Cip".obiekt[#nr].procedura := 0;
	            
	    END_CASE;
	    
	    CASE "Cip".obiekt[#nr].procedura OF
	    2:
	    //wyzwolenie timerków
	    "Cip".obiekt[#nr].SetReset.czasDoSet := 1;
	    "Cip".obiekt[#nr].SetReset.inSet :=
	    NOT "Cip".obiekt["Cip".tor[0].zbiornikWodyWtórnej.czujnikGórnegoPoziomu].hmiPotwWysterowania
	    // AND (#aktualnyKrokMycia = 5 OR #aktualnyKrokMycia = 6); // nie wiem czy to było dobrze w Orle 1
	    ;
	    "Cip".obiekt[#nr].SetReset.czasDoReset := 1;
	    "Cip".obiekt[#nr].SetReset.inReset :=
	    "Cip".obiekt["Cip".tor[0].zbiornikWodyWtórnej.czujnikGórnegoPoziomu].hmiPotwWysterowania
	    // OR (#aktualnyKrokMycia <> 5 AND #aktualnyKrokMycia <> 6);
	     ;
	    // ;
	    //załaczanie
	    "Cip".obiekt[#nr].inStartAuto := "Cip".obiekt[#nr].SetReset.wyjście;
	    
	    
	    END_CASE;
	    END_REGION
	    
	    REGION ZAWOR WYDAWCZY ŁUGU
	    
	        #nr := "Cip".tor[1].zawórWydawczyŁugu;
	        CASE "Tor1_program".program.numerKroku OF
	            7240..7243,7411,7412:
	                "Cip".obiekt[#nr].procedura := 2;
	            7100:
	                "Cip".obiekt[#nr].procedura := 3;
	            7320:
	                "Cip".obiekt[#nr].procedura := 4;
	            ELSE
	                "Cip".obiekt[#nr].procedura := 0;
	                
	        END_CASE;
	        
	    CASE "Cip".obiekt[#nr].procedura OF
	    2:
	    //wyzwolenie timerków
	    "Cip".obiekt[#nr].SetReset.czasDoSet := 3;
	    "Cip".obiekt[#nr].SetReset.inSet :=
	    "Cip".obiekt["Cip".tor[0].zbiornikŁugu.czujnikDolnegoPoziomu].hmiPotwWysterowania
	    AND (#aktualnyKrokMycia = 3);
	    
	    "Cip".obiekt[#nr].SetReset.czasDoReset := 10;
	    "Cip".obiekt[#nr].SetReset.inReset :=
	    NOT "Cip".obiekt["Cip".tor[0].zbiornikŁugu.czujnikDolnegoPoziomu].hmiPotwWysterowania
	    OR (#aktualnyKrokMycia <> 3);
	    //załaczanie
	    "Cip".obiekt[#nr].inStartAuto := "Cip".obiekt[#nr].SetReset.wyjście;
	    3:
	    //wyzwolenie timerków
	    "Cip".obiekt[#nr].SetReset.czasDoSet := 3;
	    "Cip".obiekt[#nr].SetReset.inSet :=
	    ("Tor2_program".program.numerKroku >= 7430 AND
	    "Tor2_program".program.numerKroku <= 7440);
	    
	    
	    "Cip".obiekt[#nr].SetReset.czasDoReset := 3;
	    "Cip".obiekt[#nr].SetReset.inReset :=
	    NOT ("Tor2_program".program.numerKroku >= 7430 AND
	    "Tor2_program".program.numerKroku <= 7440);
	    
	    //załaczanie
	    "Cip".obiekt[#nr].inStartAuto := "Cip".obiekt[#nr].SetReset.wyjście;
	    
	    4:
	    //wyzwolenie timerków
	    "Cip".obiekt[#nr].SetReset.czasDoSet := 3;
	    "Cip".obiekt[#nr].SetReset.inSet :=
	    "Cip".obiekt["Cip".tor[0].zbiornikŁugu.czujnikGórnegoPoziomu].hmiPotwWysterowania
	    AND (#aktualnyKrokMycia = 3);
	    
	    
	    
	    "Cip".obiekt[#nr].SetReset.czasDoReset := 3;
	    "Cip".obiekt[#nr].SetReset.inReset :=
	    NOT "Cip".obiekt["Cip".tor[0].zbiornikŁugu.czujnikGórnegoPoziomu].hmiPotwWysterowania
	    OR (#aktualnyKrokMycia <> 3);
	    
	    //załaczanie
	    "Cip".obiekt[#nr].inStartAuto := "Cip".obiekt[#nr].SetReset.wyjście;
	    
	    
	    
	    
	    
	    
	    
	    
	    END_CASE;
	    END_REGION
	    
	    REGION ZAWÓR POWROTNY ŁUGU
	    
	        #nr := "Cip".tor[1].zawórPowrotnyŁugu;
	        CASE "Tor1_program".program.numerKroku OF
	            7431,7432,7434,7435,7440:
	                "Cip".obiekt[#nr].procedura := 1;
	            7242, 7245, 7246, 7321:
	                "Cip".obiekt[#nr].procedura := 2;
	            7100:
	                "Cip".obiekt[#nr].procedura := 3;
	            7243, 7244, 7310, 7320:
	                "Cip".obiekt[#nr].procedura := 4;
	            ELSE
	                "Cip".obiekt[#nr].procedura := 0;
	        END_CASE;
	        
	    CASE "Cip".obiekt[#nr].procedura OF
	    2:
	    //wyzwolenie timerków
	    "Cip".obiekt[#nr].SetReset.czasDoSet := 1;
	    "Cip".obiekt[#nr].SetReset.inSet :=
	    "Cip".obiekt["Cip".tor[1].przewodnośćNaPowrocie].WartośćPomiaru >=
	    "Tor1_RecepturyStacjaMycia".Receptura[#aktualnyNumerReceptury].Krok[#aktualnyKrokMycia].PM[10]
	    AND (#aktualnyKrokMycia = 3)
	    AND NOT "Cip".obiekt["Cip".tor[0].zbiornikŁugu.czujnikGórnegoPoziomu].hmiPotwWysterowania;
	    
	    "Cip".obiekt[#nr].SetReset.czasDoReset := 1;
	    "Cip".obiekt[#nr].SetReset.inReset :=
	    "Cip".obiekt["Cip".tor[1].przewodnośćNaPowrocie].WartośćPomiaru <
	    "Tor1_RecepturyStacjaMycia".Receptura[#aktualnyNumerReceptury].Krok[#aktualnyKrokMycia].PM[10]
	    OR (#aktualnyKrokMycia <> 3)
	    OR "Cip".obiekt["Cip".tor[0].zbiornikŁugu.czujnikGórnegoPoziomu].hmiPotwWysterowania;
	    //załaczanie
	    "Cip".obiekt[#nr].inStartAuto := "Cip".obiekt[#nr].SetReset.wyjście;
	    3:
	    //wyzwolenie timerków
	    "Cip".obiekt[#nr].SetReset.czasDoSet := 3;
	    "Cip".obiekt[#nr].SetReset.inSet :=
	    "Cip".obiekt["Cip".tor[2].zawórWydawczyŁugu].inStartAuto
	    AND ("Tor2_program".program.numerKroku > 7400
	    AND "Tor2_program".program.numerKroku < 7470);
	    
	    
	    "Cip".obiekt[#nr].SetReset.czasDoReset := 3;
	    "Cip".obiekt[#nr].SetReset.inReset :=
	    NOT "Cip".obiekt["Cip".tor[2].zawórWydawczyŁugu].inStartAuto
	    OR ("Tor2_program".program.numerKroku < 7400
	    OR "Tor2_program".program.numerKroku > 7470);
	    
	    //załaczanie
	    "Cip".obiekt[#nr].inStartAuto := "Cip".obiekt[#nr].SetReset.wyjście;
	    
	    4:
	    //wyzwolenie timerków
	    "Cip".obiekt[#nr].SetReset.czasDoSet := 3;
	    "Cip".obiekt[#nr].SetReset.inSet :=
	    (#aktualnyKrokMycia = 3);
	    
	    "Cip".obiekt[#nr].SetReset.czasDoReset := 10;
	    "Cip".obiekt[#nr].SetReset.inReset :=
	    (#aktualnyKrokMycia <> 3);
	    //załaczanie
	    "Cip".obiekt[#nr].inStartAuto := "Cip".obiekt[#nr].SetReset.wyjście;
	    END_CASE;
	    
	    END_REGION
	    
	    REGION ZAWÓR WYDAWCZY KWASU
	        
	        #nr := "Cip".tor[1].zawórWydawczyKwasu;
	        CASE "Tor1_program".program.numerKroku OF
	            7240..7243, 7411, 7412, 7434, 7435:
	                "Cip".obiekt[#nr].procedura := 2;
	            7100:
	                "Cip".obiekt[#nr].procedura := 3;
	            7320:
	                "Cip".obiekt[#nr].procedura := 4;
	            ELSE
	                "Cip".obiekt[#nr].procedura := 0;
	                
	        END_CASE;
	        
	        CASE "Cip".obiekt[#nr].procedura OF
	            2:
	                //wyzwolenie timerków
	                "Cip".obiekt[#nr].SetReset.czasDoSet := 3;
	                "Cip".obiekt[#nr].SetReset.inSet :=
	                "Cip".obiekt["Cip".tor[0].zbiornikKwasu.czujnikDolnegoPoziomu].hmiPotwWysterowania
	                AND (#aktualnyKrokMycia = 4);
	                
	                "Cip".obiekt[#nr].SetReset.czasDoReset := 10;
	                "Cip".obiekt[#nr].SetReset.inReset :=
	                NOT "Cip".obiekt["Cip".tor[0].zbiornikKwasu.czujnikDolnegoPoziomu].hmiPotwWysterowania
	                OR (#aktualnyKrokMycia <> 4);
	                
	                //załaczanie
	                "Cip".obiekt[#nr].inStartAuto := "Cip".obiekt[#nr].SetReset.wyjście;
	            3:
	                //wyzwolenie timerków
	                "Cip".obiekt[#nr].SetReset.czasDoSet := 3;
	                "Cip".obiekt[#nr].SetReset.inSet :=
	                ("Tor2_program".program.numerKroku >= 7450 AND
	                "Tor2_program".program.numerKroku <= 7470);
	                
	                
	                "Cip".obiekt[#nr].SetReset.czasDoReset := 3;
	                "Cip".obiekt[#nr].SetReset.inReset :=
	                NOT ("Tor2_program".program.numerKroku >= 7450 AND
	                "Tor2_program".program.numerKroku <= 7470);
	                
	                //załaczanie
	                "Cip".obiekt[#nr].inStartAuto := "Cip".obiekt[#nr].SetReset.wyjście;
	                
	                
	            4:
	                //wyzwolenie timerków
	                "Cip".obiekt[#nr].SetReset.czasDoSet := 3;
	                "Cip".obiekt[#nr].SetReset.inSet :=
	                "Cip".obiekt["Cip".tor[0].zbiornikKwasu.czujnikGórnegoPoziomu].hmiPotwWysterowania
	                AND (#aktualnyKrokMycia = 4);
	                
	                
	                
	                "Cip".obiekt[#nr].SetReset.czasDoReset := 3;
	                "Cip".obiekt[#nr].SetReset.inReset :=
	                NOT "Cip".obiekt["Cip".tor[0].zbiornikKwasu.czujnikGórnegoPoziomu].hmiPotwWysterowania
	                OR (#aktualnyKrokMycia <> 4);
	                
	                //załaczanie
	                "Cip".obiekt[#nr].inStartAuto := "Cip".obiekt[#nr].SetReset.wyjście;
	                
	        END_CASE;
	    END_REGION
	    
	    REGION ZAWÓR POWROTNY KWASU
	    
	        #nr := "Cip".tor[1].zawórPowrotnyKwasu;
	        
	        CASE "Tor1_program".program.numerKroku OF
	            7460:
	                "Cip".obiekt[#nr].procedura := 1;
	            7242, 7245, 7246, 7321:
	                "Cip".obiekt[#nr].procedura := 2;
	            7100:
	                "Cip".obiekt[#nr].procedura := 3;
	            7243, 7244, 7310, 7320:
	                "Cip".obiekt[#nr].procedura := 4;
	            ELSE
	                "Cip".obiekt[#nr].procedura := 0;
	        END_CASE;
	        
	    CASE "Cip".obiekt[#nr].procedura OF
	    2:
	    //wyzwolenie timerków
	    "Cip".obiekt[#nr].SetReset.czasDoSet := 1;
	    "Cip".obiekt[#nr].SetReset.inSet :=
	    "Cip".obiekt["Cip".tor[1].przewodnośćNaPowrocie].WartośćPomiaru >=
	    "Tor1_RecepturyStacjaMycia".Receptura[#aktualnyNumerReceptury].Krok[#aktualnyKrokMycia].PM[10]
	    AND (#aktualnyKrokMycia = 4)
	    AND NOT "Cip".obiekt["Cip".tor[0].zbiornikKwasu.czujnikGórnegoPoziomu].hmiPotwWysterowania;
	    
	    "Cip".obiekt[#nr].SetReset.czasDoReset := 1;
	    "Cip".obiekt[#nr].SetReset.inReset :=
	    "Cip".obiekt["Cip".tor[1].przewodnośćNaPowrocie].WartośćPomiaru <
	    "Tor1_RecepturyStacjaMycia".Receptura[#aktualnyNumerReceptury].Krok[#aktualnyKrokMycia].PM[10]
	    OR (#aktualnyKrokMycia <> 4)
	    OR "Cip".obiekt["Cip".tor[0].zbiornikKwasu.czujnikGórnegoPoziomu].hmiPotwWysterowania;
	    //załaczanie
	    "Cip".obiekt[#nr].inStartAuto := "Cip".obiekt[#nr].SetReset.wyjście;
	    3:
	    //wyzwolenie timerków
	    "Cip".obiekt[#nr].SetReset.czasDoSet := 3;
	    "Cip".obiekt[#nr].SetReset.inSet :=
	    "Cip".obiekt["Cip".tor[2].zawórWydawczyKwasu].inStartAuto AND
	    ("Tor2_program".program.numerKroku >= 7400 AND
	    "Tor2_program".program.numerKroku <= 7470);
	    ;
	    
	    
	    "Cip".obiekt[#nr].SetReset.czasDoReset := 3;
	    "Cip".obiekt[#nr].SetReset.inReset :=
	    NOT "Cip".obiekt["Cip".tor[2].zawórWydawczyKwasu].inStartAuto
	    OR ("Tor2_program".program.numerKroku < 7400 OR
	    "Tor2_program".program.numerKroku > 7470);
	    ;
	    
	    //załaczanie
	    "Cip".obiekt[#nr].inStartAuto := "Cip".obiekt[#nr].SetReset.wyjście;
	    4:
	    //wyzwolenie timerków
	    "Cip".obiekt[#nr].SetReset.czasDoSet := 3;
	    "Cip".obiekt[#nr].SetReset.inSet := (#aktualnyKrokMycia = 4);
	    
	    "Cip".obiekt[#nr].SetReset.czasDoReset := 10;
	    "Cip".obiekt[#nr].SetReset.inReset := (#aktualnyKrokMycia <> 4);
	    
	    //załaczanie
	    "Cip".obiekt[#nr].inStartAuto := "Cip".obiekt[#nr].SetReset.wyjście;
	    END_CASE;
	    END_REGION
	    
	    REGION ZAWÓR WYDAWCZY WODY CZYSTEJ
	    
	        #nr := "Cip".tor[1].zawórWydawczyWodyCzystej;
	        
	        CASE "Tor1_program".program.numerKroku OF
	            7220..7230, 7411, 7412:
	                "Cip".obiekt[#nr].procedura := 2;
	            7244..7270, 7321, 7402, 7403, 7414, 7420, 7431, 7432, 7440, 7460:
	                "Cip".obiekt[#nr].procedura := 3;
	            7242, 7243:
	                "Cip".obiekt[#nr].procedura := 4;
	            7310, 7320:
	                "Cip".obiekt[#nr].procedura := 5;
	            7281..7291:
	                "Cip".obiekt[#nr].procedura := 6;
	            ELSE
	                "Cip".obiekt[#nr].procedura := 0;
	                
	        END_CASE;
	        
	        
	    CASE "Cip".obiekt[#nr].procedura OF
	    2:
	    //wyzwolenie timerków
	    "Cip".obiekt[#nr].SetReset.czasDoSet := 3;
	    "Cip".obiekt[#nr].SetReset.inSet :=
	    "Cip".obiekt["Cip".tor[0].zbiornikwodyCzystej.czujnikDolnegoPoziomu].hmiPotwWysterowania
	    AND NOT "Cip".obiekt["Cip".tor[0].zbiornikWodyWtórnej.czujnikDolnegoPoziomu].hmiPotwWysterowania;
	    
	    "Cip".obiekt[#nr].SetReset.czasDoReset := 10;
	    "Cip".obiekt[#nr].SetReset.inReset :=
	    NOT "Cip".obiekt["Cip".tor[0].zbiornikwodyCzystej.czujnikDolnegoPoziomu].hmiPotwWysterowania
	    OR "Cip".obiekt["Cip".tor[0].zbiornikWodyWtórnej.czujnikDolnegoPoziomu].hmiPotwWysterowania;
	    //załaczanie
	    "Cip".obiekt[#nr].inStartAuto := "Cip".obiekt[#nr].SetReset.wyjście;
	    3:
	    //wyzwolenie timerków
	    "Cip".obiekt[#nr].SetReset.czasDoSet := 3;
	    "Cip".obiekt[#nr].SetReset.inSet :=
	    "Cip".obiekt["Cip".tor[0].zbiornikwodyCzystej.czujnikDolnegoPoziomu].hmiPotwWysterowania;
	    
	    
	    "Cip".obiekt[#nr].SetReset.czasDoReset := 3;
	    "Cip".obiekt[#nr].SetReset.inReset :=
	    NOT "Cip".obiekt["Cip".tor[0].zbiornikwodyCzystej.czujnikDolnegoPoziomu].hmiPotwWysterowania;
	    
	    //załaczanie
	    "Cip".obiekt[#nr].inStartAuto := "Cip".obiekt[#nr].SetReset.wyjście;
	    
	    4:
	    //wyzwolenie timerków
	    "Cip".obiekt[#nr].SetReset.czasDoSet := 1;
	    "Cip".obiekt[#nr].SetReset.inSet :=
	    (NOT "Cip".obiekt["Cip".tor[0].zbiornikŁugu.czujnikDolnegoPoziomu].hmiPotwWysterowania AND #aktualnyKrokMycia = 3)
	    OR (NOT "Cip".obiekt["Cip".tor[0].zbiornikKwasu.czujnikDolnegoPoziomu].hmiPotwWysterowania AND #aktualnyKrokMycia = 4);
	    
	    
	    "Cip".obiekt[#nr].SetReset.czasDoReset := 5;
	    "Cip".obiekt[#nr].SetReset.inReset :=
	    ("Cip".obiekt["Cip".tor[0].zbiornikŁugu.czujnikDolnegoPoziomu].hmiPotwWysterowania AND #aktualnyKrokMycia = 3)
	    OR ("Cip".obiekt["Cip".tor[0].zbiornikKwasu.czujnikDolnegoPoziomu].hmiPotwWysterowania AND #aktualnyKrokMycia = 4);
	    //załaczanie
	    "Cip".obiekt[#nr].inStartAuto := "Cip".obiekt[#nr].SetReset.wyjście;
	    
	    5:
	    //wyzwolenie timerków
	    "Cip".obiekt[#nr].SetReset.czasDoSet := 1;
	    "Cip".obiekt[#nr].SetReset.inSet :=
	    (NOT "Cip".obiekt["Cip".tor[0].zbiornikŁugu.czujnikGórnegoPoziomu].hmiPotwWysterowania AND #aktualnyKrokMycia = 3)
	    OR (NOT "Cip".obiekt["Cip".tor[0].zbiornikKwasu.czujnikGórnegoPoziomu].hmiPotwWysterowania AND #aktualnyKrokMycia = 4);
	    
	    
	    "Cip".obiekt[#nr].SetReset.czasDoReset := 2;
	    "Cip".obiekt[#nr].SetReset.inReset :=
	    ("Cip".obiekt["Cip".tor[0].zbiornikŁugu.czujnikGórnegoPoziomu].hmiPotwWysterowania AND #aktualnyKrokMycia = 3)
	    OR ("Cip".obiekt["Cip".tor[0].zbiornikKwasu.czujnikGórnegoPoziomu].hmiPotwWysterowania AND #aktualnyKrokMycia = 4);
	    //załaczanie
	    "Cip".obiekt[#nr].inStartAuto := "Cip".obiekt[#nr].SetReset.wyjście;
	6:
	    //wyzwolenie timerków
	    "Cip".obiekt[#nr].SetReset.czasDoSet :=1;
	    "Cip".obiekt[#nr].SetReset.inSet :=
	    NOT ("Cip".obiekt["Cip".tor[1].zawórWydawczyDezynfekantu].hmiPotwWysterowania);
	    
	    
	    "Cip".obiekt[#nr].SetReset.czasDoReset := 2;
	    "Cip".obiekt[#nr].SetReset.inReset :=
	     ("Cip".obiekt["Cip".tor[1].zawórWydawczyDezynfekantu].hmiPotwWysterowania);;
	    //załaczanie
	    "Cip".obiekt[#nr].inStartAuto := "Cip".obiekt[#nr].SetReset.wyjście;
	    
	    END_CASE;
	    END_REGION
	    
	    REGION zawór wydawczy dezynfekantu
	        
	        #nr := "Cip".tor[1].zawórWydawczyDezynfekantu;
	        CASE "Tor1_program".program.numerKroku OF
	            7282..7284:
	                "Cip".obiekt[#nr].procedura := 2;
	                
	            ELSE
	                "Cip".obiekt[#nr].procedura := 0;
	                
	        END_CASE;
	        
	        CASE "Cip".obiekt[#nr].procedura OF
	            2:
	                //wyzwolenie timerków
	                "Cip".obiekt[#nr].SetReset.czasDoSet := 2;
	                "Cip".obiekt[#nr].SetReset.inSet :=
	                "Cip".obiekt["Cip".tor[1].zbiornikDezynfekantu.poziomAnalogowy].WartośćPomiaru > 10.0;
	                
	                "Cip".obiekt[#nr].SetReset.czasDoReset := 2;
	                "Cip".obiekt[#nr].SetReset.inReset :=
	                "Cip".obiekt["Cip".tor[1].zbiornikDezynfekantu.poziomAnalogowy].WartośćPomiaru < 0.01;
	                ;
	                //załaczanie
	                "Cip".obiekt[#nr].inStartAuto := "Cip".obiekt[#nr].SetReset.wyjście;
	                
	        END_CASE;
	    END_REGION
	    
	    REGION zawór powrotny dezynfekantu
	        
	        #nr := "Cip".tor[1].zawórPowrotnyDezynfekantu;
	        CASE "Tor1_program".program.numerKroku OF
	            7281..7283:
	                "Cip".obiekt[#nr].procedura :=2;
	                
	            ELSE
	                "Cip".obiekt[#nr].procedura := 0;
	                
	        END_CASE;
	        
	        CASE "Cip".obiekt[#nr].procedura OF
	            2:
	                //wyzwolenie timerków
	                "Cip".obiekt[#nr].SetReset.czasDoSet := 5;
	                "Cip".obiekt[#nr].SetReset.inSet :=
	                NOT  "Cip".obiekt["Cip".tor[1].zbiornikDezynfekantu.czujnikGórnegoPoziomu].hmiPotwWysterowania ;
	                
	                "Cip".obiekt[#nr].SetReset.czasDoReset := 0;
	                "Cip".obiekt[#nr].SetReset.inReset :=
	              "Cip".obiekt["Cip".tor[1].zbiornikDezynfekantu.czujnikGórnegoPoziomu].hmiPotwWysterowania;
	                ;
	                //załaczanie
	                "Cip".obiekt[#nr].inStartAuto := "Cip".obiekt[#nr].SetReset.wyjście;
	                
	        END_CASE;
	    END_REGION
	    
	    REGION zawór stopowy dezynfekantu
	        
	        #nr := "Cip".tor[1].zawórStopowyPowrotuDezynfekantu;
	        CASE "Tor1_program".program.numerKroku OF
	            7281..7283:
	                "Cip".obiekt[#nr].procedura := 2;
	                
	            ELSE
	                "Cip".obiekt[#nr].procedura := 0;
	                
	        END_CASE;
	        
	        CASE "Cip".obiekt[#nr].procedura OF
	            2:
	                //wyzwolenie timerków
	                "Cip".obiekt[#nr].SetReset.czasDoSet := 0;
	                "Cip".obiekt[#nr].SetReset.inSet :=
	                "Cip".obiekt["Cip".tor[1].zawórPowrotnyDezynfekantu].hmiPotwWysterowania;
	                
	                "Cip".obiekt[#nr].SetReset.czasDoReset := 0;
	                "Cip".obiekt[#nr].SetReset.inReset :=
	                NOT "Cip".obiekt["Cip".tor[1].zawórPowrotnyDezynfekantu].hmiPotwWysterowania;
	                ;
	                //załaczanie
	                "Cip".obiekt[#nr].inStartAuto := "Cip".obiekt[#nr].SetReset.wyjście;
	                
	        END_CASE;
	    END_REGION
	    
	    REGION ZAWÓR PAROWY REGULACYJNY
	    
	        #nr := "Cip".tor[1].zawórParowyRegulacyjny;
	        
	    CASE "Tor1_program".program.numerKroku OF
	    7220, 7250, 7403, 7414, 7432:
	    "Cip".obiekt[#nr].procedura := 2;
	    7242..7246, 7320, 7321, 7411, 7412, 7434, 7435:
	    "Cip".obiekt[#nr].procedura := 3;
	    
	    ELSE
	    "Cip".obiekt[#nr].procedura := 0;
	    
	    END_CASE;
	    
	    
	    CASE "Cip".obiekt[#nr].procedura OF
	    2:
	    //wyzwolenie timerków
	    "Cip".obiekt[#nr].SetReset.czasDoSet := 2;
	    "Cip".obiekt[#nr].SetReset.inSet := "Cip".obiekt["Cip".tor[1].zawórParowyOdcinający].outStartUrządzenie;
	    
	    "Cip".obiekt[#nr].SetReset.czasDoReset := 2;
	    "Cip".obiekt[#nr].SetReset.inReset := NOT "Cip".obiekt["Cip".tor[1].zawórParowyOdcinający].outStartUrządzenie;
	    
	    
	    //załaczanie
	    "Cip".obiekt[#nr].inStartAuto := "Cip".obiekt[#nr].SetReset.wyjście;
	    
	    //wysterowanie
	    "Cip".obiekt[#nr].inZadaneWysterowanieAuto :=  //pid_out wypełniamy w wywołaniu pida z out pida
	    LIMIT(IN := "Cip".obiekt[#nr].pid_Out, MN := 0.0, MX := 100.0);//pid_out ;
	    
	    ////PID
	    "Cip".obiekt[#nr].pid_SP :=
	    "Tor1_RecepturyStacjaMycia".Receptura[#aktualnyNumerReceptury].Krok[#aktualnyKrokMycia].PM[14];
	    "Cip".obiekt[#nr].pid_PV := "Cip".obiekt["Cip".tor[1].temperaturaZaWymiennikiem].WartośćPomiaru;
	    3:
	    //wyzwolenie timerków
	    "Cip".obiekt[#nr].SetReset.czasDoSet := 2;
	    "Cip".obiekt[#nr].SetReset.inSet := "Cip".obiekt["Cip".tor[1].zawórParowyOdcinający].outStartUrządzenie;
	    
	    "Cip".obiekt[#nr].SetReset.czasDoReset := 2;
	    "Cip".obiekt[#nr].SetReset.inReset := NOT "Cip".obiekt["Cip".tor[1].zawórParowyOdcinający].outStartUrządzenie;
	    
	    
	    //załaczanie
	    "Cip".obiekt[#nr].inStartAuto := "Cip".obiekt[#nr].SetReset.wyjście;
	    
	    //wysterowanie
	    "Cip".obiekt[#nr].inZadaneWysterowanieAuto :=  //pid_out wypełniamy w wywołaniu pida z out pida
	    LIMIT(IN := "Cip".obiekt[#nr].pid_Out, MN := 0.0, MX := 100.0);//pid_out ;
	    
	    ////PID
	    "Cip".obiekt[#nr].pid_SP :=
	    "Tor1_RecepturyStacjaMycia".Receptura[#aktualnyNumerReceptury].Krok[#aktualnyKrokMycia].PM[13];
	    "Cip".obiekt[#nr].pid_PV := "Cip".obiekt["Cip".tor[1].temperaturaZaWymiennikiem].WartośćPomiaru;
	    
	    0:
	    ;
	    
	    // resetowanie całkującej części regulatora aby nie przejebać temperatury
	    // "PID_Compact23".IntegralResetMode := 3;
	    // "PID_Compact23".OverwriteInitialOutputValue := "F1.SP"."203"- 1.0;
	    // "PID_Compact23".Reset := "F1".obiekt["F100LT01"].WartośćPomiaru > 70.0;
	    // := LIMIT(IN := "APA".obiekt["PID123"].outWysterowanieUrządzenia,
	    // MN := 0.0, MX := "APA".obiekt["H101TT01"].WartośćPomiaru + "H1.STP"."214");
	    
	    END_CASE;
	    
	    IF "Cip".obiekt[#nr].procedura > 0 THEN
	    
	    IF "Cip".obiekt[#nr].inStartAuto = 0 THEN
	    "Cip".obiekt[#nr].inZadaneWysterowanieAuto := 0.0;
	    "Cip".obiekt[#nr].pid_SP := 0.0;
	    END_IF;
	    END_IF;
	    
	    
	    "PID.zawórRegulacyjnyParyTor1"(Setpoint := "Cip".obiekt[#nr].pid_SP,
	                           Input := "Cip".obiekt[#nr].pid_PV,
	                           Reset := "Cip".obiekt[#nr].hmiResetAwaria,
	                           Output => "Cip".obiekt[#nr].pid_Out);
	    "PID.zawórRegulacyjnyParyTor1".Retain.CtrlParams.Gain := 1.0;
	    "PID.zawórRegulacyjnyParyTor1".Retain.CtrlParams.Ti := "Cip".obiekt[#nr].pid_I;
	    "PID.zawórRegulacyjnyParyTor1".Retain.CtrlParams.Td := "Cip".obiekt[#nr].pid_D;
	END_REGION
	
	    REGION ZAWOR PAROWY ODCINAJACY
	        
	        #nr := "Cip".tor[1].zawórParowyOdcinający;
	        CASE "Tor1_program".program.numerKroku OF
	            7220, 7240, 7242,7243, 7246, 7250, 7320, 7321, 7403, 7411, 7412, 7414, 7432, 7434, 7435:
	                "Cip".obiekt[#nr].procedura := 2;
	                
	            ELSE
	                "Cip".obiekt[#nr].procedura := 0;
	                
	        END_CASE;
	        
	        CASE "Cip".obiekt[#nr].procedura OF
	            2:
	                //wyzwolenie timerków
	                "Cip".obiekt[#nr].SetReset.czasDoSet := 2;
	                "Cip".obiekt[#nr].SetReset.inSet :=
	                "Cip".obiekt["Cip".tor[1].pompaPodawaniaCip].hmiPotwWysterowania
	                AND "Cip".obiekt["Cip".tor[1].temperaturaZaWymiennikiem].WartośćPomiaru < 90;
	                
	                "Cip".obiekt[#nr].SetReset.czasDoReset := 2;
	                "Cip".obiekt[#nr].SetReset.inReset :=
	                NOT "Cip".obiekt["Cip".tor[1].pompaPodawaniaCip].hmiPotwWysterowania
	                OR "Cip".obiekt["Cip".tor[1].temperaturaZaWymiennikiem].WartośćPomiaru >= 95;
	                //załaczanie
	                "Cip".obiekt[#nr].inStartAuto := "Cip".obiekt[#nr].SetReset.wyjście;
	        END_CASE;
	    END_REGION
	            
END_FUNCTION

FUNCTION "Tor1.procedury_sygnałów" : Void
{ S7_Optimized_Access := 'TRUE' }
VERSION : 0.1
   VAR_TEMP 
      x : Int;
      y : Int;
      numerProcedury : Int;
      indexKroku : Int;
      numerObiektu : Int;
      aktualnyNumerReceptury : Int;
      aktualnyKrokMycia : Int;
   END_VAR

   VAR CONSTANT 
      "1" : Int := 1;
      CIP2 : Int := 2;
      CIP3 : Int := 3;
      TANK_CIP : Int := 4;
      READY1 : Int := 5;
      READY2 : Int := 6;
      READY3 : Int := 7;
      CONF1 : Int := 8;
      CONF2 : Int := 9;
      ERR : Int := 10;
      PULLOUT1 : Int := 11;
      PULLOUT2 : Int := 12;
      PULLOUT3 : Int := 13;
      WATER1 : Int := 14;
      WATER2 : Int := 15;
      WATER3 : Int := 16;
      OUT1 : Int := 17;
      OUT2 : Int := 18;
      OUT3 : Int := 19;
      CONNECT1 : Int := 20;
      CONNECT2 : Int := 21;
      CONNECT3 : Int := 22;
      WHEY : Int := 23;
      AG : Int := 24;
      PUMP : Int := 25;
      FLIP : Int := 26;
      S1_RUNNING : Int := 27;
      S1_FEED : Int := 28;
      S1_START : Int := 29;
      S1_REMOTE : Int := 30;
      S1_RINSING : Int := 31;
      S1_ERR : Int := 32;
      S1_OUT : Int := 33;
   END_VAR


BEGIN
	
	// //=============================================================================
	// // Mlekomat Sp. z o.o.// (c)Copyright (2019)
	// //-----------------------------------------------------------------------------
	// // Biblioteka: Orzeł-Piotr Kowalski
	// // Testowano za pomocą: PLCSIM Advanced v.2.0 sp1
	// // Engineering: TIA Portal 15.1
	// // Ograniczenia: (typy bloków OB, itp.)
	// // Wymagania: (sprzęt, pamięć, itp.)
	// // Funkcjonalność:  Odczytanie z tablicy  "F1.sygnały.1_99.krok" numeru procedury
	// // dla każdego sygnału "Sygnały".F[1]....   i zastosowanie oewj procedury - zgodnie
	// // z dokumentem FD od technologa
	// //----------------------------------------------------------------------------
	// // Zmiany w logu:
	// // Wersja Data Autor Data wprowadzenia zmian
	// // 01.00.00 15.03.2019 Piotr Kowalski//
	// //=============================================================================
	
	// //program zawiera procedury dla sygnałów dla procedur o numerze >1  (procedura 0 i 1 jest obsługiwana w programie FB_obsługa sygnałów)
	// //procedury wyzwalane  z progrmu TablicaProcedór dla kolejnych kroków  "F1".obiekt["F100CP01"].procedura: = 2
	// //wyzwolenie procedury zero  automatycznie  wyłącza sygnał
	// //procedura:=1   wyzwala sygnał SET -- obsługiwana jest w programie FB obsłóga sygnałów
	// //
	// //
	// //open ctrl+shift+(*)Numeric
	// //close ctrl+shift+(/)Numeric
	// //
	
	// #aktualnyNumerReceptury := "CIP1_RecepturyStacjaMycia".numerUżywanejReceptury;
	// #aktualnyKrokMycia := "CIP1_RecepturyStacjaMycia".numerKrokuMycia;
	
	
	
	
	
	
	// CASE "CIP1_sygnały".sygnał[#"1"].procedura OF
	        
	//     2:
	//         IF "CIP1_RecepturyStacjaMycia".Receptura[#aktualnyNumerReceptury].Krok[#aktualnyKrokMycia].PM[21] = 1 THEN
	//             IF
	//                 ("CIP1_RecepturyStacjaMycia".Receptura[#aktualnyNumerReceptury].Krok[#aktualnyKrokMycia].PM[24] = 2101
	//                 AND "SIG".SIG[2101]=1)
	//                 OR ("CIP1_RecepturyStacjaMycia".Receptura[#aktualnyNumerReceptury].Krok[#aktualnyKrokMycia].PM[24] = 2102
	//                 AND "SIG".SIG[2102]=1)
	//                 OR ("CIP1_RecepturyStacjaMycia".Receptura[#aktualnyNumerReceptury].Krok[#aktualnyKrokMycia].PM[24] = 3101
	//                 AND "SIG".SIG[3101]=1)
	//                 OR ("CIP1_RecepturyStacjaMycia".Receptura[#aktualnyNumerReceptury].Krok[#aktualnyKrokMycia].PM[24] = 3102
	//                 AND "SIG".SIG[3102]=1)
	//                 OR ("CIP1_RecepturyStacjaMycia".Receptura[#aktualnyNumerReceptury].Krok[#aktualnyKrokMycia].PM[24] = 9401
	//                 AND "SIG".SIG[9401]=1)
	//                 OR ("CIP1_RecepturyStacjaMycia".Receptura[#aktualnyNumerReceptury].Krok[#aktualnyKrokMycia].PM[24] = 9501
	//                 AND "SIG".SIG[9501]=1)
	//                 OR ("CIP1_RecepturyStacjaMycia".Receptura[#aktualnyNumerReceptury].Krok[#aktualnyKrokMycia].PM[24] = 4101
	//                 AND "SIG".SIG[4101]=1)
	//             THEN
	//                 "CIP1_sygnały".sygnał[#"1"].inStart := 1;
	//             END_IF;
	//             ;
	//         END_IF;
	//     0:
	//         "CIP1_sygnały".sygnał[#"1"].inStart := 0;
	        
	// END_CASE;
	// "SIG".SIG[7101] := BOOL_TO_INT("CIP1_sygnały".sygnał[#"1"].inStart);
	
	// CASE "CIP1_sygnały".sygnał[#OUT1].procedura OF
	        
	//     2:
	        
	      
	//         "CIP1_sygnały".sygnał[#OUT1].inStart := "CIP1_obiekty".obiekt["C101AV13"].outStartUrządzenie;
	    
	//         ;
	//     0:
	//         "CIP1_sygnały".sygnał[#OUT1].inStart := 0;
	        
	// END_CASE;
	// "SIG".SIG[7120] := BOOL_TO_INT("CIP1_sygnały".sygnał[#OUT1].inStart);
	
	
	// CASE "CIP1_sygnały".sygnał[#AG].procedura OF
	        
	//     2:
	//         "Flipaj_cip1_sygnał_AG"(ile_petli := 999,
	//                                 czas_ON   := 100,
	//                                 czas_OFF  := 600);
	        
	        
	//         IF "CIP1_RecepturyStacjaMycia".Receptura[#aktualnyNumerReceptury].Krok[#aktualnyKrokMycia].PM[23]=1 THEN
	//             "Flipaj_cip1_sygnał_AG".in := 1;
	//             "CIP1_sygnały".sygnał[#AG].inStart := "Flipaj_cip1_sygnał_AG".Q;
	//         ELSE
	//             "Flipaj_cip1_sygnał_AG".in := 0;
	//         END_IF;
	//     0:
	//         "Flipaj_cip1_sygnał_AG".in := 0;
	//         "CIP1_sygnały".sygnał[#AG].inStart := 0;
	// END_CASE;
	// "SIG".SIG[7127] := BOOL_TO_INT("CIP1_sygnały".sygnał[#AG].inStart);
	
	
	// CASE "CIP1_sygnały".sygnał[#FLIP].procedura OF
	        
	//     2:
	//         "Flipaj_cip1_sygnał_FLIP"(ile_petli := 999,
	//                                 czas_ON   := 300,
	//                                 czas_OFF  := 600);
	        
	        
	//       // IF "CIP1_RecepturyStacjaMycia".Receptura[#aktualnyNumerReceptury].Krok[#aktualnyKrokMycia].PM[23] = 1
	//           IF 1=1
	//       THEN
	//             "Flipaj_cip1_sygnał_FLIP".in := 1;
	//             "CIP1_sygnały".sygnał[#FLIP].inStart := "Flipaj_cip1_sygnał_FLIP".Q;
	//         ELSE
	//             "Flipaj_cip1_sygnał_FLIP".in := 0;
	//         END_IF;
	//     0:
	     
	//         "CIP1_sygnały".sygnał[#FLIP].inStart := 0;
	//         "Flipaj_cip1_sygnał_FLIP"(in:=0,
	//                                   ile_petli := 999,
	//                                   czas_ON := 300,
	//                                   czas_OFF := 600);
	// END_CASE;
	// "SIG".SIG[7128] := BOOL_TO_INT("CIP1_sygnały".sygnał[#FLIP].inStart);
	
	
	// CASE "CIP1_sygnały".sygnał[#PUMP].procedura OF
	        
	//     2:
	        
	        
	//         IF "CIP1_RecepturyStacjaMycia".Receptura[#aktualnyNumerReceptury].Krok[#aktualnyKrokMycia].PM[23] = 1
	//             AND "licznik_1" < "CIP1_RecepturyStacjaMycia".Receptura[#aktualnyNumerReceptury].Krok[#aktualnyKrokMycia].PM[9] * 10
	//         THEN
	//             "licznik_1" := "licznik_1" + 1;
	//             IF "licznik_1" >= "CIP1_RecepturyStacjaMycia".Receptura[#aktualnyNumerReceptury].Krok[#aktualnyKrokMycia].PM[9] * 10
	//             THEN
	//                 "CIP1_sygnały".sygnał[#PUMP].inStart := 1;
	//             END_IF;
	            
	//         END_IF;
	//     0:
	//         "CIP1_sygnały".sygnał[#PUMP].inStart := 0;
	//         "licznik_1" := 0;
	// END_CASE;
	// "SIG".SIG[7129] := BOOL_TO_INT("CIP1_sygnały".sygnał[#PUMP].inStart);
	
	
	
	// IF "CIP1_hmi".button.bPauza.set THEN
	//     "SIG".SIG[7127] := 0;
	//     "SIG".SIG[7128] := 0;
	//     "SIG".SIG[7129] := 0;
	// END_IF;
	
	
	// "SIG".SIG[7161] := "CIP1_program".program.numerKroku;
	
	// //s1.rinsing
	// IF "CIP1_program".program.numerKroku = 7210
	//     OR "CIP1_program".program.numerKroku = 7220
	//     OR "CIP1_program".program.numerKroku = 7250
	//     OR "CIP1_program".program.numerKroku = 7270
	//     OR "CIP1_program".program.numerKroku = 7282
	    
	// THEN
	//     "SIG".SIG[7134] := 1;
	// ELSE
	//     "SIG".SIG[7134] := 0;
	// END_IF;
	// //s1.out
	// IF ("CIP1_program".program.numerKroku >= 7240
	//     AND "CIP1_program".program.numerKroku <= 7246)
	//     OR "CIP1_program".program.numerKroku = 7280
	//     OR "CIP1_program".program.numerKroku = 7281
	    
	    
	// THEN
	//     "SIG".SIG[7136] := 1;
	// ELSE
	//     "SIG".SIG[7136] := 0;
	// END_IF;
	    
	
	
	
	
	
	
	
	
END_FUNCTION

FUNCTION "Tor2.aMAIN" : Void
{ S7_Optimized_Access := 'TRUE' }
VERSION : 0.1

BEGIN
	//ponizsze FC należy napisać dla każdego urządzenia od nowa
	"Tor2.kroki"();
	"Tor2.procedury_alarmow"();
	"Tor2.procedury_obiektów"();
	"Tor2.procedury_sygnałów"();
	"Tor2_RecepturyStacjaMycia"();
	
	
	
	
	
	
	
	
	
END_FUNCTION

FUNCTION "Tor2.kroki" : Void
{ S7_Optimized_Access := 'TRUE' }
VERSION : 0.1
   VAR_TEMP 
      fdsf : Int;
      doSkasowania : Int;
      aktualnyNumerReceptury : Int;
      aktualnyKrokMycia : Int;
      sygnały_S1_czujnik_S1M1ZS02 : Bool;
   END_VAR


BEGIN
	    #aktualnyNumerReceptury := "Tor2_RecepturyStacjaMycia".numerUżywanejReceptury;
	    #aktualnyKrokMycia := "Tor2_RecepturyStacjaMycia".numerKrokuMycia;
	    "Tor2_program".program.numerKrMycia := "Tor2_RecepturyStacjaMycia".numerKrokuMycia;
	    "linia1_pompa_zezwolenie" := 1;
	    
	
	    
	    IF
	        "Tor2_hmi".button.bStop.set = 1
	        // OR "diSAFETY"=0
	    THEN
	        "Tor2_program".program.numerKroku :=7100;
	        "Tor2_hmi".button.bStop.set := 0;
	        "Tor2_hmi".button.bStart.set := 0;
	        "Tor2_hmi".button.bProdukcja.set := 0;
	        "Tor2_hmi".button.bPrzygotowanie.set := 0;
	        "Tor2_hmi".button.bPullout.set := 0;
	        "Tor2_hmi".button.bCyrkulacja.set := 0;
	        "Tor2_hmi".button.bFlux.set := 0;
	        "Tor2_hmi".button.bCip.set := 0;
	    END_IF;
	    
	    
	    "Tor2_hmi".button.bStop.kolor := BOOL_TO_INT("Tor2_hmi".button.bStop.set);
	    "Tor2_hmi".button.bStart.kolor:= BOOL_TO_INT("Tor2_hmi".button.bStart.set) ;
	    "Tor2_hmi".button.bProdukcja.kolor := BOOL_TO_INT("Tor2_hmi".button.bProdukcja.set) ;
	    "Tor2_hmi".button.bPrzygotowanie.kolor := BOOL_TO_INT("Tor2_hmi".button.bPrzygotowanie.set);
	    "Tor2_hmi".button.bPullout.kolor :=BOOL_TO_INT("Tor2_hmi".button.bPullout.set) ;
	    "Tor2_hmi".button.bCyrkulacja.kolor := BOOL_TO_INT("Tor2_hmi".button.bCyrkulacja.set);
	    "Tor2_hmi".button.bFlux.kolor := BOOL_TO_INT("Tor2_hmi".button.bFlux.set);
	    "Tor2_hmi".button.bCip.kolor :=BOOL_TO_INT("Tor2_hmi".button.bCip.set) ;
	    "Tor2_hmi".button.bPauza.kolor := BOOL_TO_INT("Tor2_hmi".button.bPauza.set AND "Clock_1Hz")*2;
	    
	
	    
	    
	    CASE "Tor2_program".program.numerKroku OF
	            
	        0: //inicjalizacja   
	            "IdźDoKroku"(inNumerKrokuDocelowy := 7100,
	                         inZadaneOpóżnienie   := 1,
	                         numerKroku           := "Tor2_program".program.numerKroku,
	                         opóźnienie           := "Tor2_program".program.opóżnienie,
	                         pauza:=  "Tor2_hmi".button.bPauza.set);
	            
	        7100://Postój
	            
	            "Cip".obiekt["Cip".tor[2].przepływomierzZaWymiennikiem].licznik1 := 0;
	            IF
	                "Tor2_hmi".button.bStart.set = 1
	            THEN
	                "IdźDoKroku"(inNumerKrokuDocelowy := 7200,
	                             inZadaneOpóżnienie   := 1,
	                             numerKroku           := "Tor2_program".program.numerKroku,
	                             opóźnienie           := "Tor2_program".program.opóżnienie,
	                             pauza:=  "Tor2_hmi".button.bPauza.set);
	                "Tor2_RecepturyStacjaMycia".numerKrokuMycia := 1;
	            END_IF;
	            
	            IF
	                "Tor2_hmi".button.bPrzygotowanie.set = 1
	            THEN
	                "IdźDoKroku"(inNumerKrokuDocelowy := 7300,
	                             inZadaneOpóżnienie   := 1,
	                             numerKroku           := "Tor2_program".program.numerKroku,
	                             opóźnienie           := "Tor2_program".program.opóżnienie,
	                             pauza:=  "Tor2_hmi".button.bPauza.set);
	                "Tor2_RecepturyStacjaMycia".numerKrokuMycia := 3;
	            END_IF;
	            
	            IF
	                "Tor2_hmi".button.bCip.set = 1
	            THEN
	                "IdźDoKroku"(inNumerKrokuDocelowy := 7400,
	                             inZadaneOpóżnienie := 1,
	                             numerKroku := "Tor2_program".program.numerKroku,
	                             opóźnienie := "Tor2_program".program.opóżnienie,
	                             pauza:=  "Tor2_hmi".button.bPauza.set);
	                "Tor2_RecepturyStacjaMycia".numerKrokuMycia := 1;
	            END_IF;
	            
	            "Tor2_program".program.zadana1 := 0;
	            "Tor2_program".program.aktualna1 := 0;
	            "Tor2_program".program.zadana2 := 0;
	            "Tor2_program".program.aktualna2 := 0;
	           
	            
	            
	            
	        7200://Zaczytanie numeru receptury (program ustawia Krok mycia =1)
	            
	            IF "Tor2_RecepturyStacjaMycia".bPokazOknoWyboruReceptury = 0 THEN
	                "Tor2_RecepturyStacjaMycia".bPokazOknoWyboruReceptury := 1;
	            END_IF;
	            IF
	                "Tor2_RecepturyStacjaMycia".klawiszUżyjTejReceptury = 1
	            THEN
	                "IdźDoKroku"(inNumerKrokuDocelowy := 7201,
	                             inZadaneOpóżnienie := 0,
	                             numerKroku := "Tor2_program".program.numerKroku,
	                             opóźnienie := "Tor2_program".program.opóżnienie,
	                             pauza := "Tor2_hmi".button.bPauza.set);
	                "Tor2_RecepturyStacjaMycia".bPokazOknoWyboruReceptury := 0;
	               
	                #doSkasowania := 1;
	                
	
	                
	                
	            END_IF;
	            "Tor2_program".program.zadana1 := 0;
	            "Tor2_program".program.aktualna1 := 0;
	            "Tor2_program".program.zadana2 := 0;
	            "Tor2_program".program.aktualna2 := 0;
	            
	            
	            #aktualnyNumerReceptury := "Tor2_RecepturyStacjaMycia".numerWyswietlanejReceptury;
	            IF "Tor2_RecepturyStacjaMycia"."klawiszReceptura-1" OR "Tor2_RecepturyStacjaMycia"."klawiszReceptura+1" THEN
	                "Tor2_hmi".bPomińŁugowanie := NOT
	                INT_TO_BOOL("Tor2_RecepturyStacjaMycia".Receptura[#aktualnyNumerReceptury].Krok[3].PM[2]);
	                "Tor2_hmi".bPomińKwasowanie := NOT
	                INT_TO_BOOL("Tor2_RecepturyStacjaMycia".Receptura[#aktualnyNumerReceptury].Krok[4].PM[2]);
	                "Tor2_hmi".bPomińDesynfekcje := NOT
	                INT_TO_BOOL("Tor2_RecepturyStacjaMycia".Receptura[#aktualnyNumerReceptury].Krok[6].PM[2]);
	            END_IF;
	         7201: //      Potwierdzenie gotowości obiektu
	             #aktualnyNumerReceptury := #aktualnyNumerReceptury;
	             #aktualnyKrokMycia := #aktualnyKrokMycia;
	             "Tor2_RecepturyStacjaMycia".Receptura[#aktualnyNumerReceptury].Krok[#aktualnyKrokMycia].PM[23]:=
	             "Tor2_RecepturyStacjaMycia".Receptura[#aktualnyNumerReceptury].Krok[#aktualnyKrokMycia].PM[23] ;
	            // jeżeli wybrano sprawdzenie czujnika
	            IF "Tor2_RecepturyStacjaMycia".Receptura[#aktualnyNumerReceptury].Krok[#aktualnyKrokMycia].PM[21] = 1
	                //sprawdzenie czujnika dla wybranego obiektu
	            THEN
	                //jezeli wybrano obiekt do mycia numer 1234
	                IF 
	                    // "SIG".SIG[
	                    // REAL_TO_INT("Tor1_RecepturyStacjaMycia".Receptura[#aktualnyNumerReceptury].Krok[#aktualnyKrokMycia].PM[24])]=1
	                    //i jest sygnał z czujnika
	                    //AND #sygnały_S1_czujnik_S1M1ZS02 = 1
	                    //
	                    "CipSignals".Object[
	                    REAL_TO_INT("Tor2_RecepturyStacjaMycia".Receptura[#aktualnyNumerReceptury].Krok[#aktualnyKrokMycia].PM[24])].toCip.bReadyToCip=1
	                    THEN
	                    "IdźDoKroku"(inNumerKrokuDocelowy := 7202,
	                                 inZadaneOpóżnienie   := 5,
	                                 numerKroku           := "Tor2_program".program.numerKroku,
	                                 opóźnienie           := "Tor2_program".program.opóżnienie,
	                                 pauza:=  "Tor2_hmi".button.bPauza.set);
	                END_IF;
	            ELSE
	                "IdźDoKroku"(inNumerKrokuDocelowy := 7202,
	                             inZadaneOpóżnienie := 10,
	                             numerKroku := "Tor2_program".program.numerKroku,
	                             opóźnienie := "Tor2_program".program.opóżnienie,
	                             pauza := "Tor2_hmi".button.bPauza.set);
	            END_IF;
	            
	            "Tor2_program".program.zadana1 := "Tor2_RecepturyStacjaMycia".Receptura[#aktualnyNumerReceptury].Krok[#aktualnyKrokMycia].PM[23];
	            "Tor2_program".program.aktualna1 := 0;
	            "Tor2_program".program.zadana2 := "Tor2_RecepturyStacjaMycia".Receptura[#aktualnyNumerReceptury].Krok[#aktualnyKrokMycia].PM[24];
	            "Tor2_program".program.aktualna2 := BOOL_TO_INT("CipSignals".Object[
	            REAL_TO_INT("Tor2_RecepturyStacjaMycia".Receptura[#aktualnyNumerReceptury].Krok[#aktualnyKrokMycia].PM[24])].toCip.bReadyToCip);
	            
	        7202://Drenaż zbiornika
	            
	            
	            IF
	                "Cip".obiekt["Cip".tor[2].czujnikPrzepływuNaPowrocie].hmiPotwWysterowania = 1
	            THEN
	                "Tor2_program".program.opóżnienie := 0;
	            END_IF;
	            "IdźDoKroku"(inNumerKrokuDocelowy := 7210,
	                         inZadaneOpóżnienie   := "Tor2_RecepturyStacjaMycia".Receptura[#aktualnyNumerReceptury].Krok[#aktualnyKrokMycia].PM[7],
	                         numerKroku           := "Tor2_program".program.numerKroku,
	                         opóźnienie           := "Tor2_program".program.opóżnienie,
	                         pauza:=  "Tor2_hmi".button.bPauza.set);
	            
	            "Tor2_program".program.zadana1 := "Tor2_RecepturyStacjaMycia".Receptura[#aktualnyNumerReceptury].Krok[#aktualnyKrokMycia].PM[7];
	            "Tor2_program".program.aktualna1 := "Tor2_program".program.opóżnienie;
	            "Tor2_program".program.zadana2 := 0;
	            "Tor2_program".program.aktualna2 := INT_TO_REAL(BOOL_TO_INT(  "Cip".obiekt["Cip".tor[2].czujnikPrzepływuNaPowrocie].hmiPotwWysterowania = 1)) * 1.0;
	            
	            IF "Tor2_RecepturyStacjaMycia".Receptura[#aktualnyNumerReceptury].Krok[#aktualnyKrokMycia].PM[23] = 0
	            THEN
	                "Tor2_program".program.numerKroku := 7210;
	            END_IF;
	           
	            
	            
	        7210: //płukanie zimne
	            
	            IF "Tor2_RecepturyStacjaMycia".Receptura[#aktualnyNumerReceptury].Krok[#aktualnyKrokMycia].PM[2] = 0
	            THEN
	                ;
	                "Tor2_program".program.numerKroku := 7220;
	                "Tor2_RecepturyStacjaMycia".numerKrokuMycia :=
	                "Tor2_RecepturyStacjaMycia".numerKrokuMycia + 1;
	            END_IF;
	            
	            
	            ;
	            IF "Cip".obiekt["Cip".tor[2].przewodnośćNaPowrocie].WartośćPomiaru <=
	                "Tor2_RecepturyStacjaMycia".Receptura[#aktualnyNumerReceptury].Krok[#aktualnyKrokMycia].PM[12] +
	                "Tor2_RecepturyStacjaMycia".Receptura[#aktualnyNumerReceptury].Krok[#aktualnyKrokMycia].PM[14]
	            THEN
	                "Cip".obiekt["Cip".tor[2].przepływomierzZaWymiennikiem].zerujLicznik1 := 0;
	                "Cip".obiekt["Cip".tor[2].przepływomierzZaWymiennikiem].startLicznik1 := 1;
	            ELSE
	                "Cip".obiekt["Cip".tor[2].przepływomierzZaWymiennikiem].startLicznik1 := 0;
	            END_IF;
	            
	            IF "Cip".obiekt["Cip".tor[2].przepływomierzZaWymiennikiem].licznik1 >
	                "Tor2_RecepturyStacjaMycia".Receptura[#aktualnyNumerReceptury].Krok[#aktualnyKrokMycia].PM[5]
	            THEN
	                "Cip".obiekt["Cip".tor[2].przepływomierzZaWymiennikiem].zerujLicznik1 := 0;
	                "Cip".obiekt["Cip".tor[2].przepływomierzZaWymiennikiem].startLicznik1 := 0;
	                "Cip".obiekt["Cip".tor[2].przepływomierzZaWymiennikiem].licznik1 := 0;
	                "Tor2_program".program.numerKroku := 7220;
	                "Tor2_RecepturyStacjaMycia".numerKrokuMycia :=
	                "Tor2_RecepturyStacjaMycia".numerKrokuMycia + 1;
	            END_IF;
	            
	            
	            "Tor2_program".program.zadana1 := "Tor2_RecepturyStacjaMycia".Receptura[#aktualnyNumerReceptury].Krok[#aktualnyKrokMycia].PM[12] +
	            "Tor2_RecepturyStacjaMycia".Receptura[#aktualnyNumerReceptury].Krok[#aktualnyKrokMycia].PM[14];
	            "Tor2_program".program.aktualna1 := "Cip".obiekt["Cip".tor[2].przewodnośćNaPowrocie].WartośćPomiaru;
	            "Tor2_program".program.zadana2 := "Tor2_RecepturyStacjaMycia".Receptura[#aktualnyNumerReceptury].Krok[#aktualnyKrokMycia].PM[5];
	            "Tor2_program".program.aktualna2 := "Cip".obiekt["Cip".tor[2].przepływomierzZaWymiennikiem].licznik1;
	            
	        7220: //płukanie ciepłe
	            
	            IF "Tor2_RecepturyStacjaMycia".Receptura[#aktualnyNumerReceptury].Krok[#aktualnyKrokMycia].PM[2] = 0
	            THEN
	                ;
	                "Tor2_program".program.numerKroku := 7230;
	                "Tor2_RecepturyStacjaMycia".numerKrokuMycia :=
	                "Tor2_RecepturyStacjaMycia".numerKrokuMycia + 1;
	            END_IF;
	            
	            
	            ;
	            IF "Cip".obiekt["Cip".tor[2].przewodnośćNaPowrocie].WartośćPomiaru <=
	                "Tor2_RecepturyStacjaMycia".Receptura[#aktualnyNumerReceptury].Krok[#aktualnyKrokMycia].PM[12] +
	                "Tor2_RecepturyStacjaMycia".Receptura[#aktualnyNumerReceptury].Krok[#aktualnyKrokMycia].PM[15]
	                AND
	                "Cip".obiekt["Cip".tor[2].temperaturaNaPowrocie].WartośćPomiaru >=
	                "Tor2_RecepturyStacjaMycia".Receptura[#aktualnyNumerReceptury].Krok[#aktualnyKrokMycia].PM[14] -
	                "Tor2_RecepturyStacjaMycia".Receptura[#aktualnyNumerReceptury].Krok[#aktualnyKrokMycia].PM[16]
	                
	            THEN
	                "Cip".obiekt["Cip".tor[2].przepływomierzZaWymiennikiem].zerujLicznik1 := 0;
	                "Cip".obiekt["Cip".tor[2].przepływomierzZaWymiennikiem].startLicznik1 := 1;
	            ELSE
	                "Cip".obiekt["Cip".tor[2].przepływomierzZaWymiennikiem].startLicznik1 := 0;
	            END_IF;
	            
	            IF "Cip".obiekt["Cip".tor[2].przepływomierzZaWymiennikiem].licznik1 >
	                "Tor2_RecepturyStacjaMycia".Receptura[#aktualnyNumerReceptury].Krok[#aktualnyKrokMycia].PM[5]
	            THEN
	                "Cip".obiekt["Cip".tor[2].przepływomierzZaWymiennikiem].zerujLicznik1 := 0;
	                "Cip".obiekt["Cip".tor[2].przepływomierzZaWymiennikiem].startLicznik1 := 0;
	               
	                
	                "linia1_pompa_zezwolenie" := 0;
	                "IdźDoKroku"(inNumerKrokuDocelowy := 7221,
	                             inZadaneOpóżnienie := 9,
	                             numerKroku := "Tor2_program".program.numerKroku,
	                             opóźnienie := "Tor2_program".program.opóżnienie,
	                             pauza := "Tor2_hmi".button.bPauza.set);
	                
	                // "CIP1_RecepturyStacjaMycia".numerKrokuMycia :=
	                // "CIP1_RecepturyStacjaMycia".numerKrokuMycia + 1;
	            END_IF;
	            
	            
	            "Tor2_program".program.zadana1 := "Tor2_RecepturyStacjaMycia".Receptura[#aktualnyNumerReceptury].Krok[#aktualnyKrokMycia].PM[14] -
	            "Tor2_RecepturyStacjaMycia".Receptura[#aktualnyNumerReceptury].Krok[#aktualnyKrokMycia].PM[16];
	            "Tor2_program".program.aktualna1 := "Cip".obiekt["Cip".tor[2].temperaturaNaPowrocie].WartośćPomiaru;
	            "Tor2_program".program.zadana2 := "Tor2_RecepturyStacjaMycia".Receptura[#aktualnyNumerReceptury].Krok[#aktualnyKrokMycia].PM[5];
	            "Tor2_program".program.aktualna2 := "Cip".obiekt["Cip".tor[2].przepływomierzZaWymiennikiem].licznik1;
	            
	            
	        7221:
	            "Cip".obiekt["Cip".tor[2].przepływomierzZaWymiennikiem].licznik1 := 0;
	            "Tor2_RecepturyStacjaMycia".numerKrokuMycia :=
	            "Tor2_RecepturyStacjaMycia".numerKrokuMycia + 1;
	            "Tor2_program".program.numerKroku := 7230;
	            
	            
	        7230://sprawdzenie kroku mycia)
	            
	            IF
	                "Tor2_RecepturyStacjaMycia".numerKrokuMycia < 5
	            THEN
	                "IdźDoKroku"(inNumerKrokuDocelowy := 7240,
	                             inZadaneOpóżnienie   := 1,
	                             numerKroku           := "Tor2_program".program.numerKroku,
	                             opóźnienie           := "Tor2_program".program.opóżnienie,
	                             pauza:=  "Tor2_hmi".button.bPauza.set);
	            END_IF;
	            IF
	                "Tor2_RecepturyStacjaMycia".numerKrokuMycia >= 5
	            THEN
	                "IdźDoKroku"(inNumerKrokuDocelowy := 7270,
	                             inZadaneOpóżnienie   := 1,
	                             numerKroku           := "Tor2_program".program.numerKroku,
	                             opóźnienie           := "Tor2_program".program.opóżnienie,
	                             pauza:=  "Tor2_hmi".button.bPauza.set);
	                "Tor2_hmi".button.bCip.set := 0;
	            END_IF;
	            "Tor2_program".program.zadana1 := 0;
	            "Tor2_program".program.aktualna1 := 0;
	            "Tor2_program".program.zadana2 := 0;
	            "Tor2_program".program.aktualna2 := 0;
	            
	        7240://Wypełnienie linii do zbiornika 
	            
	            IF "Tor2_RecepturyStacjaMycia".Receptura[#aktualnyNumerReceptury].Krok[#aktualnyKrokMycia].PM[2] = 0
	                
	                OR (#aktualnyKrokMycia=3 AND "Tor2_hmi".bPomińŁugowanie)
	                OR (#aktualnyKrokMycia=4 AND "Tor2_hmi".bPomińKwasowanie)
	                OR (#aktualnyKrokMycia=6 AND "Tor2_hmi".bPomińDesynfekcje)
	           
	                
	            THEN
	                ;
	                "Tor2_program".program.numerKroku := 7260;
	            END_IF;
	            IF "Tor2_RecepturyStacjaMycia".Receptura[#aktualnyNumerReceptury].Krok[#aktualnyKrokMycia].PM[23] = 0
	                AND "Tor2_RecepturyStacjaMycia".Receptura[#aktualnyNumerReceptury].Krok[#aktualnyKrokMycia].PM[2] =1
	            THEN
	                
	                "Cip".obiekt["Cip".tor[2].pompaPodawaniaCip].inStartAuto := 0;
	                "IdźDoKroku"(inNumerKrokuDocelowy := 7242,
	                             inZadaneOpóżnienie := 0.2,
	                             numerKroku := "Tor2_program".program.numerKroku,
	                             opóźnienie := "Tor2_program".program.opóżnienie,
	                             pauza := "Tor2_hmi".button.bPauza.set);
	            END_IF;
	            
	            "Cip".obiekt["Cip".tor[2].przepływomierzZaWymiennikiem].zerujLicznik1 := 0;
	            "Cip".obiekt["Cip".tor[2].przepływomierzZaWymiennikiem].startLicznik1 := 1;
	            
	            
	            IF "Cip".obiekt["Cip".tor[2].przepływomierzZaWymiennikiem].licznik1 >
	                "Tor2_RecepturyStacjaMycia".Receptura[#aktualnyNumerReceptury].Krok[#aktualnyKrokMycia].PM[8]
	                AND "Tor2_RecepturyStacjaMycia".Receptura[#aktualnyNumerReceptury].Krok[#aktualnyKrokMycia].PM[23] = 1
	               
	            THEN
	                "Cip".obiekt["Cip".tor[2].przepływomierzZaWymiennikiem].zerujLicznik1 := 0;
	                "Cip".obiekt["Cip".tor[2].przepływomierzZaWymiennikiem].startLicznik1 := 0;
	               
	                
	                "linia1_pompa_zezwolenie" := 0;
	                "IdźDoKroku"(inNumerKrokuDocelowy := 7239,
	                             inZadaneOpóżnienie := 9,
	                             numerKroku := "Tor2_program".program.numerKroku,
	                             opóźnienie := "Tor2_program".program.opóżnienie,
	                             pauza := "Tor2_hmi".button.bPauza.set);
	            END_IF;
	            
	            
	            
	            "Tor2_program".program.zadana1 := "Tor2_RecepturyStacjaMycia".Receptura[#aktualnyNumerReceptury].Krok[#aktualnyKrokMycia].PM[8];
	            "Tor2_program".program.aktualna1 := "Cip".obiekt["Cip".tor[2].przepływomierzZaWymiennikiem].licznik1;
	            "Tor2_program".program.zadana2 := 0;
	            "Tor2_program".program.aktualna2 := 0;
	            
	            ;
	        7239:
	            "Cip".obiekt["Cip".tor[2].przepływomierzZaWymiennikiem].licznik1 := 0;
	            "Tor2_program".program.numerKroku := 7241;
	            
	            
	            
	        7241://Drenaż zbiornika
	            
	            IF "Tor2_RecepturyStacjaMycia".Receptura[#aktualnyNumerReceptury].Krok[#aktualnyKrokMycia].PM[23] = 0
	            THEN
	                "Tor2_program".program.numerKroku := 7242;
	            END_IF;
	            
	            IF
	                "Cip".obiekt["Cip".tor[2].czujnikPrzepływuNaPowrocie].hmiPotwWysterowania = 1
	            THEN
	                "Tor2_program".program.opóżnienie := 0;
	            END_IF;
	            "IdźDoKroku"(inNumerKrokuDocelowy := 7242,
	                         inZadaneOpóżnienie   := "Tor2_RecepturyStacjaMycia".Receptura[#aktualnyNumerReceptury].Krok[#aktualnyKrokMycia].PM[7],
	                         numerKroku           := "Tor2_program".program.numerKroku,
	                         opóźnienie           := "Tor2_program".program.opóżnienie,
	                         pauza:=  "Tor2_hmi".button.bPauza.set);
	            
	            "Tor2_program".program.zadana1 := "Tor2_RecepturyStacjaMycia".Receptura[#aktualnyNumerReceptury].Krok[#aktualnyKrokMycia].PM[7];
	            "Tor2_program".program.aktualna1 := "Tor2_program".program.opóżnienie;
	            "Tor2_program".program.zadana2 := 0;
	            "Tor2_program".program.aktualna2 := INT_TO_REAL(BOOL_TO_INT("Cip".obiekt["Cip".tor[2].czujnikPrzepływuNaPowrocie].hmiPotwWysterowania = 1)) * 1.0;
	            
	            
	            
	            
	        7242: //Wypełnienie obiegu środkiem myjącym
	            
	            IF "Cip".obiekt["Cip".tor[2].przewodnośćNaPowrocie].WartośćPomiaru >=
	                "Tor2_RecepturyStacjaMycia".Receptura[#aktualnyNumerReceptury].Krok[#aktualnyKrokMycia].PM[10] -
	                "Tor2_RecepturyStacjaMycia".Receptura[#aktualnyNumerReceptury].Krok[#aktualnyKrokMycia].PM[15]
	            THEN
	                "Tor2_program".program.numerKroku := 7243;
	                
	            END_IF;
	            
	            "Tor2_program".program.zadana1 := "Tor2_RecepturyStacjaMycia".Receptura[#aktualnyNumerReceptury].Krok[#aktualnyKrokMycia].PM[10] -
	            "Tor2_RecepturyStacjaMycia".Receptura[#aktualnyNumerReceptury].Krok[#aktualnyKrokMycia].PM[15];
	            "Tor2_program".program.aktualna1 := "Cip".obiekt["Cip".tor[2].przewodnośćNaPowrocie].WartośćPomiaru;
	            "Tor2_program".program.zadana2 := 0;
	            "Tor2_program".program.aktualna2 := 0;
	            
	        7243://    Odliczanie czasu mycia
	            
	            
	            IF
	                "Cip".obiekt["Cip".tor[2].przewodnośćNaPowrocie].WartośćPomiaru >=
	                "Tor2_RecepturyStacjaMycia".Receptura[#aktualnyNumerReceptury].Krok[#aktualnyKrokMycia].PM[10] -
	                "Tor2_RecepturyStacjaMycia".Receptura[#aktualnyNumerReceptury].Krok[#aktualnyKrokMycia].PM[15]
	                AND
	                "Cip".obiekt["Cip".tor[2].temperaturaNaPowrocie].WartośćPomiaru >=
	                "Tor2_RecepturyStacjaMycia".Receptura[#aktualnyNumerReceptury].Krok[#aktualnyKrokMycia].PM[13] -
	                "Tor2_RecepturyStacjaMycia".Receptura[#aktualnyNumerReceptury].Krok[#aktualnyKrokMycia].PM[16]
	            THEN
	                ;
	            ELSE
	                "Tor2_program".program.opóżnienie := "Tor2_program".program.opóżnienie -0.1;
	            END_IF;
	            "IdźDoKroku"(inNumerKrokuDocelowy := 7244,
	                         inZadaneOpóżnienie   := "Tor2_RecepturyStacjaMycia".Receptura[#aktualnyNumerReceptury].Krok[#aktualnyKrokMycia].PM[6],
	                         numerKroku           := "Tor2_program".program.numerKroku,
	                         opóźnienie           := "Tor2_program".program.opóżnienie,
	                         pauza:=  "Tor2_hmi".button.bPauza.set);
	            
	            
	            
	            "Tor2_program".program.zadana1 := "Tor2_RecepturyStacjaMycia".Receptura[#aktualnyNumerReceptury].Krok[#aktualnyKrokMycia].PM[13] -
	            "Tor2_RecepturyStacjaMycia".Receptura[#aktualnyNumerReceptury].Krok[#aktualnyKrokMycia].PM[16];
	            "Tor2_program".program.aktualna1 := "Cip".obiekt["Cip".tor[2].temperaturaNaPowrocie].WartośćPomiaru;
	            "Tor2_program".program.zadana2 := "Tor2_RecepturyStacjaMycia".Receptura[#aktualnyNumerReceptury].Krok[#aktualnyKrokMycia].PM[6];
	            "Tor2_program".program.aktualna2 := "Tor2_program".program.opóżnienie;
	            
	            
	        7244:// Wypełnienie linii do zbiornika wodą
	            
	            
	            IF "Tor2_RecepturyStacjaMycia".Receptura[#aktualnyNumerReceptury].Krok[#aktualnyKrokMycia].PM[23] = 0
	            THEN
	                "Tor2_program".program.numerKroku := 7246;
	            END_IF;
	            
	            "Cip".obiekt["Cip".tor[2].przepływomierzZaWymiennikiem].zerujLicznik1 := 0;
	            "Cip".obiekt["Cip".tor[2].przepływomierzZaWymiennikiem].startLicznik1 := 1;
	            
	            
	            IF "Cip".obiekt["Cip".tor[2].przepływomierzZaWymiennikiem].licznik1 >
	                "Tor2_RecepturyStacjaMycia".Receptura[#aktualnyNumerReceptury].Krok[#aktualnyKrokMycia].PM[8]
	            THEN
	                "Cip".obiekt["Cip".tor[2].przepływomierzZaWymiennikiem].zerujLicznik1 := 0;
	                "Cip".obiekt["Cip".tor[2].przepływomierzZaWymiennikiem].startLicznik1 := 0;
	                "Cip".obiekt["Cip".tor[2].przepływomierzZaWymiennikiem].licznik1 := 0;
	                "Tor2_program".program.numerKroku := 7245;
	            END_IF;
	            
	            
	            
	            "Tor2_program".program.zadana1 := "Tor2_RecepturyStacjaMycia".Receptura[#aktualnyNumerReceptury].Krok[#aktualnyKrokMycia].PM[8];
	            "Tor2_program".program.aktualna1 := "Cip".obiekt["Cip".tor[2].przepływomierzZaWymiennikiem].licznik1;
	            "Tor2_program".program.zadana2 := 0;
	            "Tor2_program".program.aktualna2 := 0;
	            
	            
	        7245: //Drenaż zbiornika
	            IF "Tor2_RecepturyStacjaMycia".Receptura[#aktualnyNumerReceptury].Krok[#aktualnyKrokMycia].PM[23] = 0
	            THEN
	                "Tor2_program".program.numerKroku := 7246;
	            END_IF;
	            
	            IF
	                "Cip".obiekt["Cip".tor[2].czujnikPrzepływuNaPowrocie].hmiPotwWysterowania = 1
	            THEN
	                "Tor2_program".program.opóżnienie := 0;
	            END_IF;
	            "IdźDoKroku"(inNumerKrokuDocelowy := 7246,
	                         inZadaneOpóżnienie   := "Tor2_RecepturyStacjaMycia".Receptura[#aktualnyNumerReceptury].Krok[#aktualnyKrokMycia].PM[7],
	                         numerKroku           := "Tor2_program".program.numerKroku,
	                         opóźnienie           := "Tor2_program".program.opóżnienie,
	                         pauza:=  "Tor2_hmi".button.bPauza.set);
	            
	            "Tor2_program".program.zadana1 := "Tor2_RecepturyStacjaMycia".Receptura[#aktualnyNumerReceptury].Krok[#aktualnyKrokMycia].PM[7];
	            "Tor2_program".program.aktualna1 := "Tor2_program".program.opóżnienie;
	            "Tor2_program".program.zadana2 := 0;
	            "Tor2_program".program.aktualna2 := INT_TO_REAL(BOOL_TO_INT("Cip".obiekt["Cip".tor[2].czujnikPrzepływuNaPowrocie].hmiPotwWysterowania = 1)) * 1.0;
	            
	        7246://             Zawracanie środka myjącego
	            
	            IF "Cip".obiekt["Cip".tor[2].przewodnośćNaPowrocie].WartośćPomiaru<
	                "Tor2_RecepturyStacjaMycia".Receptura[#aktualnyNumerReceptury].Krok[#aktualnyKrokMycia].PM[10] +
	                "Tor2_RecepturyStacjaMycia".Receptura[#aktualnyNumerReceptury].Krok[#aktualnyKrokMycia].PM[15]
	            THEN
	                "IdźDoKroku"(inNumerKrokuDocelowy := 7250,
	                             inZadaneOpóżnienie := 3,
	                             numerKroku := "Tor2_program".program.numerKroku,
	                             opóźnienie := "Tor2_program".program.opóżnienie,
	                             pauza:=  "Tor2_hmi".button.bPauza.set);
	                
	            END_IF;
	            IF "Cip".obiekt["Cip".tor[2].przewodnośćNaPowrocie].WartośćPomiaru >
	                "Tor2_RecepturyStacjaMycia".Receptura[#aktualnyNumerReceptury].Krok[#aktualnyKrokMycia].PM[10] +
	                "Tor2_RecepturyStacjaMycia".Receptura[#aktualnyNumerReceptury].Krok[#aktualnyKrokMycia].PM[15]
	            THEN
	                "Tor2_program".program.opóżnienie := 0;
	            END_IF;
	       
	            
	            "Tor2_program".program.zadana1 := "Tor2_RecepturyStacjaMycia".Receptura[#aktualnyNumerReceptury].Krok[#aktualnyKrokMycia].PM[10] +
	            "Tor2_RecepturyStacjaMycia".Receptura[#aktualnyNumerReceptury].Krok[#aktualnyKrokMycia].PM[15];
	            "Tor2_program".program.aktualna1 := "Cip".obiekt["Cip".tor[2].przewodnośćNaPowrocie].WartośćPomiaru;
	            "Tor2_program".program.zadana2 := 0;
	            "Tor2_program".program.aktualna2 := 0;
	            
	            
	        7250://    Płukanie międzyfazowe
	            
	            IF
	                "Cip".obiekt["Cip".tor[2].przewodnośćNaPowrocie].WartośćPomiaru <
	                "Tor2_RecepturyStacjaMycia".Receptura[#aktualnyNumerReceptury].Krok[#aktualnyKrokMycia].PM[12] +
	                "Tor2_RecepturyStacjaMycia".Receptura[#aktualnyNumerReceptury].Krok[#aktualnyKrokMycia].PM[15]
	                AND
	                "Cip".obiekt["Cip".tor[2].temperaturaNaPowrocie].WartośćPomiaru >=
	                "Tor2_RecepturyStacjaMycia".Receptura[#aktualnyNumerReceptury].Krok[#aktualnyKrokMycia].PM[14] -
	                "Tor2_RecepturyStacjaMycia".Receptura[#aktualnyNumerReceptury].Krok[#aktualnyKrokMycia].PM[16]
	            THEN
	                "Cip".obiekt["Cip".tor[2].przepływomierzZaWymiennikiem].zerujLicznik1 := 0;
	                "Cip".obiekt["Cip".tor[2].przepływomierzZaWymiennikiem].startLicznik1 := 1;
	            ELSE
	                "Cip".obiekt["Cip".tor[2].przepływomierzZaWymiennikiem].startLicznik1 := 0;
	            END_IF;
	            
	            
	            IF "Cip".obiekt["Cip".tor[2].przepływomierzZaWymiennikiem].licznik1 >
	                "Tor2_RecepturyStacjaMycia".Receptura[#aktualnyNumerReceptury].Krok[#aktualnyKrokMycia].PM[5]
	            THEN
	                "Cip".obiekt["Cip".tor[2].przepływomierzZaWymiennikiem].zerujLicznik1 := 0;
	                "Cip".obiekt["Cip".tor[2].przepływomierzZaWymiennikiem].startLicznik1 := 0;
	               
	                
	                "linia1_pompa_zezwolenie" := 0;
	                "IdźDoKroku"(inNumerKrokuDocelowy := 7251,
	                             inZadaneOpóżnienie := 0,
	                             numerKroku := "Tor2_program".program.numerKroku,
	                             opóźnienie := "Tor2_program".program.opóżnienie,
	                             pauza := "Tor2_hmi".button.bPauza.set);
	            END_IF;
	            
	            "Tor2_program".program.zadana1 := "Tor2_RecepturyStacjaMycia".Receptura[#aktualnyNumerReceptury].Krok[#aktualnyKrokMycia].PM[14] -
	            "Tor2_RecepturyStacjaMycia".Receptura[#aktualnyNumerReceptury].Krok[#aktualnyKrokMycia].PM[16];
	            "Tor2_program".program.aktualna1 := "Cip".obiekt["Cip".tor[2].temperaturaNaPowrocie].WartośćPomiaru;
	            "Tor2_program".program.zadana2 := "Tor2_RecepturyStacjaMycia".Receptura[#aktualnyNumerReceptury].Krok[#aktualnyKrokMycia].PM[5];
	            "Tor2_program".program.aktualna2 := "Cip".obiekt["Cip".tor[2].przepływomierzZaWymiennikiem].licznik1;
	            
	        7251:
	            
	        
	            "Tor2_program".program.numerKroku := 7260;
	            
	            "Cip".obiekt["Cip".tor[2].przepływomierzZaWymiennikiem].licznik1 := 0;
	            
	        7260://KONIEC MYCIA
	            
	            "IdźDoKroku"(inNumerKrokuDocelowy := 7230,
	                         inZadaneOpóżnienie   := 0,
	                         numerKroku           := "Tor2_program".program.numerKroku,
	                         opóźnienie           := "Tor2_program".program.opóżnienie,
	                         pauza:=  "Tor2_hmi".button.bPauza.set);
	            "Tor2_RecepturyStacjaMycia".numerKrokuMycia :=
	            "Tor2_RecepturyStacjaMycia".numerKrokuMycia + 1;
	            "Tor2_program".program.zadana1 := 0;
	            "Tor2_program".program.aktualna1 := 0;
	            "Tor2_program".program.zadana2 := 10;
	            "Tor2_program".program.aktualna2 := "Tor2_program".program.opóżnienie;
	            
	        7270://Płukanie główne
	            
